LIN {X 0,Y 626.002,Z 844.06,A -85,B 0,C 180,E1 6698.138,E2 6698.138} C_VEL
LIN {X 0,Y 626.101,Z 844.06,A -85,B 0,C 180,E1 6703.663,E2 6703.663} C_VEL
LIN {X 0,Y 628.264,Z 852.739,A -85,B 0,C 180,E1 6704.183,E2 6704.183} C_VEL
LIN {X 0,Y 630.269,Z 865.489,A -85,B 0,C 180,E1 6704.573,E2 6704.573} C_VEL
LIN {X 0,Y 651.429,Z 905.185,A -85,B 0,C 180,E1 6707.05,E2 6707.05} C_VEL
LIN {X 0,Y 646.579,Z 984.33,A -85,B 0,C 180,E1 6708.978,E2 6708.978} C_VEL
LIN {X 0,Y 639.779,Z 1059.441,A -85,B 0,C 180,E1 6712.384,E2 6712.384} C_VEL
LIN {X 0,Y 632.449,Z 1127.06,A -85,B 0,C 180,E1 6717.105,E2 6717.105} C_VEL
LIN {X 0,Y 626.29,Z 1184.219,A -85,B 0,C 180,E1 6722.849,E2 6722.849} C_VEL
LIN {X 0,Y 621.93,Z 1231.471,A -85,B 0,C 180,E1 6729.651,E2 6729.651} C_VEL
LIN {X 0,Y 619.696,Z 1263.198,A -85,B 0,C 180,E1 6736.556,E2 6736.556} C_VEL
LIN {X 0,Y 619.192,Z 1280.004,A -85,B 0,C 180,E1 6742.684,E2 6742.684} C_VEL
LIN {X 0,Y 619.266,Z 1286.38,A -85,B 0,C 180,E1 6747.895,E2 6747.895} C_VEL
LIN {X 0,Y 619.049,Z 1283.806,A -85,B 0,C 180,E1 6754.919,E2 6754.919} C_VEL
LIN {X 0,Y 619.245,Z 1270.708,A -85,B 0,C 180,E1 6761.153,E2 6761.153} C_VEL
LIN {X 0,Y 620.48,Z 1246.742,A -85,B 0,C 180,E1 6767.407,E2 6767.407} C_VEL
LIN {X 0,Y 623.202,Z 1210.805,A -85,B 0,C 180,E1 6773.673,E2 6773.673} C_VEL
LIN {X 0,Y 628.657,Z 1158.622,A -85,B 0,C 180,E1 6779.994,E2 6779.994} C_VEL
LIN {X 0,Y 635.99,Z 1095.052,A -85,B 0,C 180,E1 6785.36,E2 6785.36} C_VEL
LIN {X 0,Y 643.433,Z 1024.758,A -85,B 0,C 180,E1 6789.381,E2 6789.381} C_VEL
LIN {X 0,Y 649.249,Z 949.588,A -85,B 0,C 180,E1 6792.052,E2 6792.052} C_VEL
LIN {X 0,Y 650.101,Z 899.28,A -85,B 0,C 180,E1 6793.162,E2 6793.162} C_VEL
LIN {X 0,Y 618.004,Z 844.06,A -85,B 0,C 180,E1 6797.103,E2 6797.103} C_VEL
LIN {X 0,Y 618.586,Z 844.06,A -85,B 0,C 180,E1 6805.214,E2 6805.214} C_VEL
LIN {X 0,Y 618.31,Z 844.06,A -85,B 0,C 180,E1 6814.598,E2 6814.598} C_VEL
LIN {X 0,Y 618.343,Z 844.06,A -85,B 0,C 180,E1 6823.636,E2 6823.636} C_VEL
LIN {X 0,Y 618.382,Z 844.06,A -85,B 0,C 180,E1 6832.269,E2 6832.269} C_VEL
LIN {X 0,Y 618.586,Z 844.06,A -85,B 0,C 180,E1 6839.32,E2 6839.32} C_VEL
LIN {X 0,Y 618.554,Z 844.06,A -85,B 0,C 180,E1 6846.805,E2 6846.805} C_VEL
LIN {X 0,Y 618.35,Z 844.06,A -85,B 0,C 180,E1 6854.951,E2 6854.951} C_VEL
LIN {X 0,Y 618.062,Z 844.06,A -85,B 0,C 180,E1 6863.054,E2 6863.054} C_VEL
LIN {X 0,Y 617.97,Z 844.06,A -85,B 0,C 180,E1 6871.883,E2 6871.883} C_VEL
LIN {X 0,Y 617.773,Z 844.06,A -85,B 0,C 180,E1 6880.628,E2 6880.628} C_VEL
LIN {X 0,Y 618.221,Z 845.887,A -85,B 0,C 180,E1 6883.215,E2 6883.215} C_VEL
LIN {X 0,Y 651.122,Z 903.195,A -85,B 0,C 180,E1 6887.124,E2 6887.124} C_VEL
LIN {X 0,Y 646.443,Z 978.639,A -85,B 0,C 180,E1 6889.093,E2 6889.093} C_VEL
LIN {X 0,Y 639.82,Z 1050.163,A -85,B 0,C 180,E1 6892.387,E2 6892.387} C_VEL
LIN {X 0,Y 632.376,Z 1116.636,A -85,B 0,C 180,E1 6897.018,E2 6897.018} C_VEL
LIN {X 0,Y 625.899,Z 1175.076,A -85,B 0,C 180,E1 6902.89,E2 6902.89} C_VEL
LIN {X 0,Y 621.742,Z 1219.649,A -85,B 0,C 180,E1 6909.287,E2 6909.287} C_VEL
LIN {X 0,Y 619.652,Z 1249.811,A -85,B 0,C 180,E1 6915.601,E2 6915.601} C_VEL
LIN {X 0,Y 619.132,Z 1267.73,A -85,B 0,C 180,E1 6921.549,E2 6921.549} C_VEL
LIN {X 0,Y 618.746,Z 1276.413,A -85,B 0,C 180,E1 6927.893,E2 6927.893} C_VEL
LIN {X 0,Y 619.029,Z 1275.319,A -85,B 0,C 180,E1 6933.511,E2 6933.511} C_VEL
LIN {X 0,Y 619.043,Z 1264.068,A -85,B 0,C 180,E1 6939.874,E2 6939.874} C_VEL
LIN {X 0,Y 619.898,Z 1243.034,A -85,B 0,C 180,E1 6945.975,E2 6945.975} C_VEL
LIN {X 0,Y 622.4,Z 1209.021,A -85,B 0,C 180,E1 6952.378,E2 6952.378} C_VEL
LIN {X 0,Y 627.314,Z 1160.484,A -85,B 0,C 180,E1 6958.696,E2 6958.696} C_VEL
LIN {X 0,Y 634.383,Z 1098.839,A -85,B 0,C 180,E1 6964.31,E2 6964.31} C_VEL
LIN {X 0,Y 642.002,Z 1029.13,A -85,B 0,C 180,E1 6968.645,E2 6968.645} C_VEL
LIN {X 0,Y 648.194,Z 955.723,A -85,B 0,C 180,E1 6971.557,E2 6971.557} C_VEL
LIN {X 0,Y 649.534,Z 900.272,A -85,B 0,C 180,E1 6972.971,E2 6972.971} C_VEL
LIN {X 0,Y 618.229,Z 844.06,A -85,B 0,C 180,E1 6976.947,E2 6976.947} C_VEL
LIN {X 0,Y 618.186,Z 844.06,A -85,B 0,C 180,E1 6985.268,E2 6985.268} C_VEL
LIN {X 0,Y 618.232,Z 844.06,A -85,B 0,C 180,E1 6993.554,E2 6993.554} C_VEL
LIN {X 0,Y 618.387,Z 844.06,A -85,B 0,C 180,E1 7002.119,E2 7002.119} C_VEL
LIN {X 0,Y 619.238,Z 844.06,A -85,B 0,C 180,E1 7009.389,E2 7009.389} C_VEL
LIN {X 0,Y 619.236,Z 844.06,A -85,B 0,C 180,E1 7017.871,E2 7017.871} C_VEL
LIN {X 0,Y 618.571,Z 844.06,A -85,B 0,C 180,E1 7026.817,E2 7026.817} C_VEL
LIN {X 0,Y 618.341,Z 844.06,A -85,B 0,C 180,E1 7034.904,E2 7034.904} C_VEL
LIN {X 0,Y 618.093,Z 844.06,A -85,B 0,C 180,E1 7043.061,E2 7043.061} C_VEL
LIN {X 0,Y 618.015,Z 844.06,A -85,B 0,C 180,E1 7051.827,E2 7051.827} C_VEL
LIN {X 0,Y 617.714,Z 844.06,A -85,B 0,C 180,E1 7060.572,E2 7060.572} C_VEL
LIN {X 0,Y 618.172,Z 845.961,A -85,B 0,C 180,E1 7063.102,E2 7063.102} C_VEL
LIN {X 0,Y 630.269,Z 865.489,A -85,B 0,C 180,E1 7064.573,E2 7064.573} C_VEL
LIN {X 0,Y 639.982,Z 896.297,A -85,B 0,C 180,E1 7065.929,E2 7065.929} C_VEL
LIN {X 0,Y 645.504,Z 909.832,A -85,B 0,C 180,E1 7066.642,E2 7066.642} C_VEL
LIN {X 0,Y 640.268,Z 987.254,A -85,B 0,C 180,E1 7068.602,E2 7068.602} C_VEL
LIN {X 0,Y 633.06,Z 1061.429,A -85,B 0,C 180,E1 7072.041,E2 7072.041} C_VEL
LIN {X 0,Y 625.297,Z 1128.203,A -85,B 0,C 180,E1 7076.784,E2 7076.784} C_VEL
LIN {X 0,Y 618.672,Z 1185.973,A -85,B 0,C 180,E1 7082.704,E2 7082.704} C_VEL
LIN {X 0,Y 614.273,Z 1231.129,A -85,B 0,C 180,E1 7089.327,E2 7089.327} C_VEL
LIN {X 0,Y 611.806,Z 1263.197,A -85,B 0,C 180,E1 7096.38,E2 7096.38} C_VEL
LIN {X 0,Y 611.195,Z 1280.147,A -85,B 0,C 180,E1 7102.667,E2 7102.667} C_VEL
LIN {X 0,Y 611.278,Z 1286.38,A -85,B 0,C 180,E1 7107.867,E2 7107.867} C_VEL
LIN {X 0,Y 611.058,Z 1283.803,A -85,B 0,C 180,E1 7114.983,E2 7114.983} C_VEL
LIN {X 0,Y 611.24,Z 1270.149,A -85,B 0,C 180,E1 7121.495,E2 7121.495} C_VEL
LIN {X 0,Y 612.589,Z 1246.769,A -85,B 0,C 180,E1 7127.632,E2 7127.632} C_VEL
LIN {X 0,Y 615.51,Z 1210.805,A -85,B 0,C 180,E1 7133.987,E2 7133.987} C_VEL
LIN {X 0,Y 621.262,Z 1160.127,A -85,B 0,C 180,E1 7140.23,E2 7140.23} C_VEL
LIN {X 0,Y 629.016,Z 1096.867,A -85,B 0,C 180,E1 7145.672,E2 7145.672} C_VEL
LIN {X 0,Y 636.904,Z 1027.182,A -85,B 0,C 180,E1 7149.738,E2 7149.738} C_VEL
LIN {X 0,Y 643.085,Z 952.285,A -85,B 0,C 180,E1 7152.469,E2 7152.469} C_VEL
LIN {X 0,Y 644.166,Z 902.371,A -85,B 0,C 180,E1 7153.604,E2 7153.604} C_VEL
LIN {X 0,Y 610.109,Z 844.06,A -85,B 0,C 180,E1 7157.763,E2 7157.763} C_VEL
LIN {X 0,Y 610.509,Z 844.06,A -85,B 0,C 180,E1 7166.321,E2 7166.321} C_VEL
LIN {X 0,Y 610.219,Z 844.06,A -85,B 0,C 180,E1 7175.109,E2 7175.109} C_VEL
LIN {X 0,Y 610.345,Z 844.06,A -85,B 0,C 180,E1 7183.415,E2 7183.415} C_VEL
LIN {X 0,Y 610.388,Z 844.06,A -85,B 0,C 180,E1 7192.167,E2 7192.167} C_VEL
LIN {X 0,Y 610.587,Z 844.06,A -85,B 0,C 180,E1 7199.311,E2 7199.311} C_VEL
LIN {X 0,Y 610.683,Z 844.06,A -85,B 0,C 180,E1 7206.442,E2 7206.442} C_VEL
LIN {X 0,Y 610.294,Z 844.06,A -85,B 0,C 180,E1 7215.153,E2 7215.153} C_VEL
LIN {X 0,Y 610.144,Z 844.06,A -85,B 0,C 180,E1 7222.693,E2 7222.693} C_VEL
LIN {X 0,Y 610.061,Z 844.06,A -85,B 0,C 180,E1 7230.949,E2 7230.949} C_VEL
LIN {X 0,Y 609.85,Z 844.06,A -85,B 0,C 180,E1 7239.4,E2 7239.4} C_VEL
LIN {X 0,Y 610.054,Z 845.695,A -85,B 0,C 180,E1 7242.388,E2 7242.388} C_VEL
LIN {X 0,Y 644.996,Z 906.338,A -85,B 0,C 180,E1 7246.69,E2 7246.69} C_VEL
LIN {X 0,Y 640.096,Z 981.944,A -85,B 0,C 180,E1 7248.736,E2 7248.736} C_VEL
LIN {X 0,Y 632.886,Z 1053.967,A -85,B 0,C 180,E1 7252.147,E2 7252.147} C_VEL
LIN {X 0,Y 624.872,Z 1120.556,A -85,B 0,C 180,E1 7256.926,E2 7256.926} C_VEL
LIN {X 0,Y 617.979,Z 1178.841,A -85,B 0,C 180,E1 7263,E2 7263} C_VEL
LIN {X 0,Y 613.578,Z 1223.371,A -85,B 0,C 180,E1 7269.673,E2 7269.673} C_VEL
LIN {X 0,Y 611.531,Z 1252.307,A -85,B 0,C 180,E1 7276.085,E2 7276.085} C_VEL
LIN {X 0,Y 611.009,Z 1269.257,A -85,B 0,C 180,E1 7282.154,E2 7282.154} C_VEL
LIN {X 0,Y 610.752,Z 1276.413,A -85,B 0,C 180,E1 7287.866,E2 7287.866} C_VEL
LIN {X 0,Y 611.052,Z 1275.32,A -85,B 0,C 180,E1 7293.557,E2 7293.557} C_VEL
LIN {X 0,Y 611.058,Z 1264.069,A -85,B 0,C 180,E1 7300.005,E2 7300.005} C_VEL
LIN {X 0,Y 611.996,Z 1243.038,A -85,B 0,C 180,E1 7306.187,E2 7306.187} C_VEL
LIN {X 0,Y 614.716,Z 1209.023,A -85,B 0,C 180,E1 7312.673,E2 7312.673} C_VEL
LIN {X 0,Y 619.887,Z 1161.231,A -85,B 0,C 180,E1 7318.988,E2 7318.988} C_VEL
LIN {X 0,Y 627.318,Z 1100.446,A -85,B 0,C 180,E1 7324.619,E2 7324.619} C_VEL
LIN {X 0,Y 635.357,Z 1031.58,A -85,B 0,C 180,E1 7328.985,E2 7328.985} C_VEL
LIN {X 0,Y 641.984,Z 958.36,A -85,B 0,C 180,E1 7331.959,E2 7331.959} C_VEL
LIN {X 0,Y 643.686,Z 903.738,A -85,B 0,C 180,E1 7333.39,E2 7333.39} C_VEL
LIN {X 0,Y 610.146,Z 844.06,A -85,B 0,C 180,E1 7337.638,E2 7337.638} C_VEL
LIN {X 0,Y 610.15,Z 844.06,A -85,B 0,C 180,E1 7346.372,E2 7346.372} C_VEL
LIN {X 0,Y 610.27,Z 844.06,A -85,B 0,C 180,E1 7355.099,E2 7355.099} C_VEL
LIN {X 0,Y 610.582,Z 844.06,A -85,B 0,C 180,E1 7363.374,E2 7363.374} C_VEL
LIN {X 0,Y 610.862,Z 844.06,A -85,B 0,C 180,E1 7370.687,E2 7370.687} C_VEL
LIN {X 0,Y 611.253,Z 844.06,A -85,B 0,C 180,E1 7377.843,E2 7377.843} C_VEL
LIN {X 0,Y 610.695,Z 844.06,A -85,B 0,C 180,E1 7386.395,E2 7386.395} C_VEL
LIN {X 0,Y 610.29,Z 844.06,A -85,B 0,C 180,E1 7395.106,E2 7395.106} C_VEL
LIN {X 0,Y 610.163,Z 844.06,A -85,B 0,C 180,E1 7402.642,E2 7402.642} C_VEL
LIN {X 0,Y 610.075,Z 844.06,A -85,B 0,C 180,E1 7410.951,E2 7410.951} C_VEL
LIN {X 0,Y 609.814,Z 844.06,A -85,B 0,C 180,E1 7419.343,E2 7419.343} C_VEL
LIN {X 0,Y 609.982,Z 845.677,A -85,B 0,C 180,E1 7422.271,E2 7422.271} C_VEL
LIN {X 0,Y 639.982,Z 896.297,A -85,B 0,C 180,E1 7425.929,E2 7425.929} C_VEL
LIN {X 0,Y 641.79,Z 912.839,A -85,B 0,C 180,E1 7426.384,E2 7426.384} C_VEL
LIN {X 0,Y 638.723,Z 931.558,A -85,B 0,C 180,E1 7426.567,E2 7426.567} C_VEL
LIN {X 0,Y 633.009,Z 1002.704,A -85,B 0,C 180,E1 7428.723,E2 7428.723} C_VEL
LIN {X 0,Y 625.002,Z 1075.016,A -85,B 0,C 180,E1 7432.413,E2 7432.413} C_VEL
LIN {X 0,Y 616.67,Z 1140.57,A -85,B 0,C 180,E1 7437.469,E2 7437.469} C_VEL
LIN {X 0,Y 609.846,Z 1195.877,A -85,B 0,C 180,E1 7443.613,E2 7443.613} C_VEL
LIN {X 0,Y 605.6,Z 1237.509,A -85,B 0,C 180,E1 7450.241,E2 7450.241} C_VEL
LIN {X 0,Y 603.548,Z 1265.683,A -85,B 0,C 180,E1 7456.93,E2 7456.93} C_VEL
LIN {X 0,Y 602.957,Z 1281.732,A -85,B 0,C 180,E1 7463.501,E2 7463.501} C_VEL
LIN {X 0,Y 602.724,Z 1286.838,A -85,B 0,C 180,E1 7469.279,E2 7469.279} C_VEL
LIN {X 0,Y 602.912,Z 1282.883,A -85,B 0,C 180,E1 7475.774,E2 7475.774} C_VEL
LIN {X 0,Y 603.311,Z 1267.998,A -85,B 0,C 180,E1 7482.337,E2 7482.337} C_VEL
LIN {X 0,Y 604.879,Z 1243.162,A -85,B 0,C 180,E1 7488.643,E2 7488.643} C_VEL
LIN {X 0,Y 608.656,Z 1204.137,A -85,B 0,C 180,E1 7495.263,E2 7495.263} C_VEL
LIN {X 0,Y 615.213,Z 1150.124,A -85,B 0,C 180,E1 7501.632,E2 7501.632} C_VEL
LIN {X 0,Y 623.548,Z 1086.517,A -85,B 0,C 180,E1 7506.84,E2 7506.84} C_VEL
LIN {X 0,Y 631.633,Z 1017.29,A -85,B 0,C 180,E1 7510.659,E2 7510.659} C_VEL
LIN {X 0,Y 637.609,Z 945.851,A -85,B 0,C 180,E1 7513.112,E2 7513.112} C_VEL
LIN {X 0,Y 638.224,Z 905.427,A -85,B 0,C 180,E1 7514.057,E2 7514.057} C_VEL
LIN {X 0,Y 602.173,Z 844.06,A -85,B 0,C 180,E1 7518.668,E2 7518.668} C_VEL
LIN {X 0,Y 602.414,Z 844.06,A -85,B 0,C 180,E1 7527.494,E2 7527.494} C_VEL
LIN {X 0,Y 602.18,Z 844.06,A -85,B 0,C 180,E1 7535.464,E2 7535.464} C_VEL
LIN {X 0,Y 602.389,Z 844.06,A -85,B 0,C 180,E1 7543.19,E2 7543.19} C_VEL
LIN {X 0,Y 602.394,Z 844.06,A -85,B 0,C 180,E1 7552.062,E2 7552.062} C_VEL
LIN {X 0,Y 602.588,Z 844.06,A -85,B 0,C 180,E1 7559.302,E2 7559.302} C_VEL
LIN {X 0,Y 602.663,Z 844.06,A -85,B 0,C 180,E1 7566.528,E2 7566.528} C_VEL
LIN {X 0,Y 602.255,Z 844.06,A -85,B 0,C 180,E1 7575.361,E2 7575.361} C_VEL
LIN {X 0,Y 602.039,Z 844.06,A -85,B 0,C 180,E1 7583.157,E2 7583.157} C_VEL
LIN {X 0,Y 602.055,Z 844.06,A -85,B 0,C 180,E1 7591.128,E2 7591.128} C_VEL
LIN {X 0,Y 601.8,Z 844.06,A -85,B 0,C 180,E1 7600.032,E2 7600.032} C_VEL
LIN {X 0,Y 601.985,Z 845.823,A -85,B 0,C 180,E1 7601.541,E2 7601.541} C_VEL
LIN {X 0,Y 638.637,Z 908.901,A -85,B 0,C 180,E1 7606.213,E2 7606.213} C_VEL
LIN {X 0,Y 633.546,Z 986.704,A -85,B 0,C 180,E1 7608.44,E2 7608.44} C_VEL
LIN {X 0,Y 625.816,Z 1058.298,A -85,B 0,C 180,E1 7611.946,E2 7611.946} C_VEL
LIN {X 0,Y 617.375,Z 1124.269,A -85,B 0,C 180,E1 7616.839,E2 7616.839} C_VEL
LIN {X 0,Y 610.298,Z 1180.481,A -85,B 0,C 180,E1 7622.854,E2 7622.854} C_VEL
LIN {X 0,Y 605.653,Z 1224.708,A -85,B 0,C 180,E1 7629.654,E2 7629.654} C_VEL
LIN {X 0,Y 603.532,Z 1253.36,A -85,B 0,C 180,E1 7636.189,E2 7636.189} C_VEL
LIN {X 0,Y 602.998,Z 1270.597,A -85,B 0,C 180,E1 7642.776,E2 7642.776} C_VEL
LIN {X 0,Y 602.834,Z 1276.848,A -85,B 0,C 180,E1 7649.279,E2 7649.279} C_VEL
LIN {X 0,Y 603.349,Z 1272.815,A -85,B 0,C 180,E1 7655.77,E2 7655.77} C_VEL
LIN {X 0,Y 604.141,Z 1254.369,A -85,B 0,C 180,E1 7663.427,E2 7663.427} C_VEL
LIN {X 0,Y 606.173,Z 1220.954,A -85,B 0,C 180,E1 7670.948,E2 7670.948} C_VEL
LIN {X 0,Y 610.986,Z 1174.739,A -85,B 0,C 180,E1 7677.778,E2 7677.778} C_VEL
LIN {X 0,Y 618.492,Z 1116.109,A -85,B 0,C 180,E1 7683.777,E2 7683.777} C_VEL
LIN {X 0,Y 626.996,Z 1048.85,A -85,B 0,C 180,E1 7688.515,E2 7688.515} C_VEL
LIN {X 0,Y 634.3,Z 974.856,A -85,B 0,C 180,E1 7691.928,E2 7691.928} C_VEL
LIN {X 0,Y 637.711,Z 906.961,A -85,B 0,C 180,E1 7693.823,E2 7693.823} C_VEL
LIN {X 0,Y 603.496,Z 848.586,A -85,B 0,C 180,E1 7698.159,E2 7698.159} C_VEL
LIN {X 0,Y 602.067,Z 844.06,A -85,B 0,C 180,E1 7698.693,E2 7698.693} C_VEL
LIN {X 0,Y 602.188,Z 844.06,A -85,B 0,C 180,E1 7707.528,E2 7707.528} C_VEL
LIN {X 0,Y 602.45,Z 844.06,A -85,B 0,C 180,E1 7717.001,E2 7717.001} C_VEL
LIN {X 0,Y 603.091,Z 844.06,A -85,B 0,C 180,E1 7726.15,E2 7726.15} C_VEL
LIN {X 0,Y 602.563,Z 844.06,A -85,B 0,C 180,E1 7734.921,E2 7734.921} C_VEL
LIN {X 0,Y 602.486,Z 844.06,A -85,B 0,C 180,E1 7742.141,E2 7742.141} C_VEL
LIN {X 0,Y 602.347,Z 844.06,A -85,B 0,C 180,E1 7749.398,E2 7749.398} C_VEL
LIN {X 0,Y 602.15,Z 844.06,A -85,B 0,C 180,E1 7756.817,E2 7756.817} C_VEL
LIN {X 0,Y 601.982,Z 844.06,A -85,B 0,C 180,E1 7764.545,E2 7764.545} C_VEL
LIN {X 0,Y 601.966,Z 844.06,A -85,B 0,C 180,E1 7772.78,E2 7772.78} C_VEL
LIN {X 0,Y 601.834,Z 845.482,A -85,B 0,C 180,E1 7781.41,E2 7781.41} C_VEL
LIN {X 0,Y 639.487,Z 909.82,A -85,B 0,C 180,E1 7786.131,E2 7786.131} C_VEL
LIN {X 0,Y 638.723,Z 931.558,A -85,B 0,C 180,E1 7786.567,E2 7786.567} C_VEL
LIN {X 0,Y 630.191,Z 965.784,A -85,B 0,C 180,E1 7786.932,E2 7786.932} C_VEL
LIN {X 0,Y 622.808,Z 1040.446,A -85,B 0,C 180,E1 7789.96,E2 7789.96} C_VEL
LIN {X 0,Y 613.795,Z 1109.857,A -85,B 0,C 180,E1 7794.409,E2 7794.409} C_VEL
LIN {X 0,Y 605.326,Z 1171.403,A -85,B 0,C 180,E1 7800.22,E2 7800.22} C_VEL
LIN {X 0,Y 599.48,Z 1220.506,A -85,B 0,C 180,E1 7806.914,E2 7806.914} C_VEL
LIN {X 0,Y 596.496,Z 1256.298,A -85,B 0,C 180,E1 7814.139,E2 7814.139} C_VEL
LIN {X 0,Y 595.561,Z 1277.621,A -85,B 0,C 180,E1 7821.212,E2 7821.212} C_VEL
LIN {X 0,Y 595.276,Z 1286.38,A -85,B 0,C 180,E1 7827.81,E2 7827.81} C_VEL
LIN {X 0,Y 595.034,Z 1283.798,A -85,B 0,C 180,E1 7835.118,E2 7835.118} C_VEL
LIN {X 0,Y 595.261,Z 1270.096,A -85,B 0,C 180,E1 7841.824,E2 7841.824} C_VEL
LIN {X 0,Y 596.849,Z 1246.047,A -85,B 0,C 180,E1 7848.271,E2 7848.271} C_VEL
LIN {X 0,Y 600.598,Z 1208.153,A -85,B 0,C 180,E1 7855.021,E2 7855.021} C_VEL
LIN {X 0,Y 607.323,Z 1156.087,A -85,B 0,C 180,E1 7861.439,E2 7861.439} C_VEL
LIN {X 0,Y 616.062,Z 1092.607,A -85,B 0,C 180,E1 7866.879,E2 7866.879} C_VEL
LIN {X 0,Y 624.759,Z 1023.36,A -85,B 0,C 180,E1 7870.876,E2 7870.876} C_VEL
LIN {X 0,Y 631.511,Z 949.245,A -85,B 0,C 180,E1 7873.53,E2 7873.53} C_VEL
LIN {X 0,Y 632.398,Z 908.725,A -85,B 0,C 180,E1 7874.508,E2 7874.508} C_VEL
LIN {X 0,Y 594.26,Z 844.06,A -85,B 0,C 180,E1 7879.65,E2 7879.65} C_VEL
LIN {X 0,Y 594.331,Z 844.06,A -85,B 0,C 180,E1 7888.739,E2 7888.739} C_VEL
LIN {X 0,Y 594.029,Z 844.06,A -85,B 0,C 180,E1 7896.708,E2 7896.708} C_VEL
LIN {X 0,Y 594.166,Z 844.06,A -85,B 0,C 180,E1 7904.474,E2 7904.474} C_VEL
LIN {X 0,Y 594.399,Z 844.06,A -85,B 0,C 180,E1 7911.955,E2 7911.955} C_VEL
LIN {X 0,Y 594.6,Z 844.06,A -85,B 0,C 180,E1 7919.293,E2 7919.293} C_VEL
LIN {X 0,Y 594.626,Z 844.06,A -85,B 0,C 180,E1 7926.616,E2 7926.616} C_VEL
LIN {X 0,Y 594.213,Z 844.06,A -85,B 0,C 180,E1 7935.574,E2 7935.574} C_VEL
LIN {X 0,Y 594.014,Z 844.06,A -85,B 0,C 180,E1 7943.345,E2 7943.345} C_VEL
LIN {X 0,Y 593.988,Z 844.06,A -85,B 0,C 180,E1 7951.599,E2 7951.599} C_VEL
LIN {X 0,Y 593.788,Z 844.737,A -85,B 0,C 180,E1 7960.619,E2 7960.619} C_VEL
LIN {X 0,Y 631.903,Z 910.624,A -85,B 0,C 180,E1 7965.667,E2 7965.667} C_VEL
LIN {X 0,Y 627.171,Z 989.671,A -85,B 0,C 180,E1 7968.064,E2 7968.064} C_VEL
LIN {X 0,Y 618.902,Z 1061.446,A -85,B 0,C 180,E1 7971.673,E2 7971.673} C_VEL
LIN {X 0,Y 609.783,Z 1128.357,A -85,B 0,C 180,E1 7976.787,E2 7976.787} C_VEL
LIN {X 0,Y 602.362,Z 1184.134,A -85,B 0,C 180,E1 7982.974,E2 7982.974} C_VEL
LIN {X 0,Y 597.785,Z 1225.778,A -85,B 0,C 180,E1 7989.584,E2 7989.584} C_VEL
LIN {X 0,Y 595.521,Z 1254.664,A -85,B 0,C 180,E1 7996.376,E2 7996.376} C_VEL
LIN {X 0,Y 595.012,Z 1270.593,A -85,B 0,C 180,E1 8002.679,E2 8002.679} C_VEL
LIN {X 0,Y 594.855,Z 1276.848,A -85,B 0,C 180,E1 8009.27,E2 8009.27} C_VEL
LIN {X 0,Y 595.372,Z 1272.905,A -85,B 0,C 180,E1 8015.785,E2 8015.785} C_VEL
LIN {X 0,Y 596.161,Z 1254.37,A -85,B 0,C 180,E1 8023.61,E2 8023.61} C_VEL
LIN {X 0,Y 598.335,Z 1221.307,A -85,B 0,C 180,E1 8031.173,E2 8031.173} C_VEL
LIN {X 0,Y 603.513,Z 1175.31,A -85,B 0,C 180,E1 8038.08,E2 8038.08} C_VEL
LIN {X 0,Y 611.38,Z 1117.449,A -85,B 0,C 180,E1 8044.1,E2 8044.1} C_VEL
LIN {X 0,Y 620.389,Z 1050.271,A -85,B 0,C 180,E1 8048.909,E2 8048.909} C_VEL
LIN {X 0,Y 628.192,Z 975.916,A -85,B 0,C 180,E1 8052.387,E2 8052.387} C_VEL
LIN {X 0,Y 631.865,Z 910.539,A -85,B 0,C 180,E1 8054.249,E2 8054.249} C_VEL
LIN {X 0,Y 597.028,Z 850.282,A -85,B 0,C 180,E1 8058.829,E2 8058.829} C_VEL
LIN {X 0,Y 594.037,Z 844.06,A -85,B 0,C 180,E1 8059.336,E2 8059.336} C_VEL
LIN {X 0,Y 594.214,Z 844.06,A -85,B 0,C 180,E1 8068.414,E2 8068.414} C_VEL
LIN {X 0,Y 594.431,Z 844.06,A -85,B 0,C 180,E1 8076.673,E2 8076.673} C_VEL
LIN {X 0,Y 595.06,Z 844.06,A -85,B 0,C 180,E1 8085.96,E2 8085.96} C_VEL
LIN {X 0,Y 594.555,Z 844.06,A -85,B 0,C 180,E1 8094.853,E2 8094.853} C_VEL
LIN {X 0,Y 594.497,Z 844.06,A -85,B 0,C 180,E1 8102.17,E2 8102.17} C_VEL
LIN {X 0,Y 594.351,Z 844.06,A -85,B 0,C 180,E1 8109.526,E2 8109.526} C_VEL
LIN {X 0,Y 594.166,Z 844.06,A -85,B 0,C 180,E1 8117.05,E2 8117.05} C_VEL
LIN {X 0,Y 593.955,Z 844.06,A -85,B 0,C 180,E1 8124.985,E2 8124.985} C_VEL
LIN {X 0,Y 593.904,Z 844.06,A -85,B 0,C 180,E1 8133.283,E2 8133.283} C_VEL
LIN {X 0,Y 593.96,Z 846.045,A -85,B 0,C 180,E1 8140.554,E2 8140.554} C_VEL
LIN {X 0,Y 631.597,Z 909.164,A -85,B 0,C 180,E1 8145.429,E2 8145.429} C_VEL
LIN {X 0,Y 633.352,Z 922.085,A -85,B 0,C 180,E1 8145.877,E2 8145.877} C_VEL
LIN {X 0,Y 630.191,Z 965.784,A -85,B 0,C 180,E1 8146.932,E2 8146.932} C_VEL
LIN {X 0,Y 621.085,Z 999.235,A -85,B 0,C 180,E1 8147.582,E2 8147.582} C_VEL
LIN {X 0,Y 612.174,Z 1072.89,A -85,B 0,C 180,E1 8151.327,E2 8151.327} C_VEL
LIN {X 0,Y 602.922,Z 1138.686,A -85,B 0,C 180,E1 8156.439,E2 8156.439} C_VEL
LIN {X 0,Y 595.243,Z 1194.536,A -85,B 0,C 180,E1 8162.726,E2 8162.726} C_VEL
LIN {X 0,Y 590.122,Z 1237.505,A -85,B 0,C 180,E1 8169.7,E2 8169.7} C_VEL
LIN {X 0,Y 587.589,Z 1266.845,A -85,B 0,C 180,E1 8176.948,E2 8176.948} C_VEL
LIN {X 0,Y 586.963,Z 1282.869,A -85,B 0,C 180,E1 8184.059,E2 8184.059} C_VEL
LIN {X 0,Y 586.597,Z 1286.838,A -85,B 0,C 180,E1 8190.741,E2 8190.741} C_VEL
LIN {X 0,Y 586.966,Z 1281.727,A -85,B 0,C 180,E1 8196.677,E2 8196.677} C_VEL
LIN {X 0,Y 587.825,Z 1264.523,A -85,B 0,C 180,E1 8203.806,E2 8203.806} C_VEL
LIN {X 0,Y 590.982,Z 1231.552,A -85,B 0,C 180,E1 8211.449,E2 8211.449} C_VEL
LIN {X 0,Y 596.367,Z 1185.929,A -85,B 0,C 180,E1 8218.413,E2 8218.413} C_VEL
LIN {X 0,Y 604.488,Z 1127.965,A -85,B 0,C 180,E1 8224.541,E2 8224.541} C_VEL
LIN {X 0,Y 613.812,Z 1060.538,A -85,B 0,C 180,E1 8229.434,E2 8229.434} C_VEL
LIN {X 0,Y 622.441,Z 986.1,A -85,B 0,C 180,E1 8232.909,E2 8232.909} C_VEL
LIN {X 0,Y 626.686,Z 912.291,A -85,B 0,C 180,E1 8234.955,E2 8234.955} C_VEL
LIN {X 0,Y 586.267,Z 844.06,A -85,B 0,C 180,E1 8240.471,E2 8240.471} C_VEL
LIN {X 0,Y 586.285,Z 844.06,A -85,B 0,C 180,E1 8247.993,E2 8247.993} C_VEL
LIN {X 0,Y 586.026,Z 844.06,A -85,B 0,C 180,E1 8256.734,E2 8256.734} C_VEL
LIN {X 0,Y 586.182,Z 844.06,A -85,B 0,C 180,E1 8264.257,E2 8264.257} C_VEL
LIN {X 0,Y 586.419,Z 844.06,A -85,B 0,C 180,E1 8271.844,E2 8271.844} C_VEL
LIN {X 0,Y 586.601,Z 844.06,A -85,B 0,C 180,E1 8279.283,E2 8279.283} C_VEL
LIN {X 0,Y 586.613,Z 844.06,A -85,B 0,C 180,E1 8286.707,E2 8286.707} C_VEL
LIN {X 0,Y 586.46,Z 844.06,A -85,B 0,C 180,E1 8294.25,E2 8294.25} C_VEL
LIN {X 0,Y 586.025,Z 844.06,A -85,B 0,C 180,E1 8303.266,E2 8303.266} C_VEL
LIN {X 0,Y 585.905,Z 844.06,A -85,B 0,C 180,E1 8312.087,E2 8312.087} C_VEL
LIN {X 0,Y 585.929,Z 845.473,A -85,B 0,C 180,E1 8319.727,E2 8319.727} C_VEL
LIN {X 0,Y 623.732,Z 909.084,A -85,B 0,C 180,E1 8324.888,E2 8324.888} C_VEL
LIN {X 0,Y 627.011,Z 921.583,A -85,B 0,C 180,E1 8325.499,E2 8325.499} C_VEL
LIN {X 0,Y 620.96,Z 991.443,A -85,B 0,C 180,E1 8327.634,E2 8327.634} C_VEL
LIN {X 0,Y 612.352,Z 1062.034,A -85,B 0,C 180,E1 8331.231,E2 8331.231} C_VEL
LIN {X 0,Y 602.741,Z 1128.788,A -85,B 0,C 180,E1 8336.393,E2 8336.393} C_VEL
LIN {X 0,Y 594.859,Z 1184.695,A -85,B 0,C 180,E1 8342.684,E2 8342.684} C_VEL
LIN {X 0,Y 590.017,Z 1225.773,A -85,B 0,C 180,E1 8349.303,E2 8349.303} C_VEL
LIN {X 0,Y 587.578,Z 1254.663,A -85,B 0,C 180,E1 8356.188,E2 8356.188} C_VEL
LIN {X 0,Y 587.03,Z 1270.589,A -85,B 0,C 180,E1 8362.578,E2 8362.578} C_VEL
LIN {X 0,Y 586.853,Z 1276.848,A -85,B 0,C 180,E1 8369.26,E2 8369.26} C_VEL
LIN {X 0,Y 587.386,Z 1272.894,A -85,B 0,C 180,E1 8375.873,E2 8375.873} C_VEL
LIN {X 0,Y 588.155,Z 1254.372,A -85,B 0,C 180,E1 8383.799,E2 8383.799} C_VEL
LIN {X 0,Y 590.474,Z 1222.359,A -85,B 0,C 180,E1 8391.271,E2 8391.271} C_VEL
LIN {X 0,Y 595.942,Z 1176.92,A -85,B 0,C 180,E1 8398.261,E2 8398.261} C_VEL
LIN {X 0,Y 604.211,Z 1119.325,A -85,B 0,C 180,E1 8404.384,E2 8404.384} C_VEL
LIN {X 0,Y 613.75,Z 1052.329,A -85,B 0,C 180,E1 8409.273,E2 8409.273} C_VEL
LIN {X 0,Y 622.012,Z 978.323,A -85,B 0,C 180,E1 8412.807,E2 8412.807} C_VEL
LIN {X 0,Y 625.949,Z 913.829,A -85,B 0,C 180,E1 8414.7,E2 8414.7} C_VEL
LIN {X 0,Y 592.883,Z 856.335,A -85,B 0,C 180,E1 8419.181,E2 8419.181} C_VEL
LIN {X 0,Y 586.013,Z 844.06,A -85,B 0,C 180,E1 8420.215,E2 8420.215} C_VEL
LIN {X 0,Y 586.197,Z 844.06,A -85,B 0,C 180,E1 8429.664,E2 8429.664} C_VEL
LIN {X 0,Y 586.413,Z 844.06,A -85,B 0,C 180,E1 8437.943,E2 8437.943} C_VEL
LIN {X 0,Y 587.197,Z 844.06,A -85,B 0,C 180,E1 8447.29,E2 8447.29} C_VEL
LIN {X 0,Y 587.239,Z 844.06,A -85,B 0,C 180,E1 8457.755,E2 8457.755} C_VEL
LIN {X 0,Y 586.612,Z 844.06,A -85,B 0,C 180,E1 8466.659,E2 8466.659} C_VEL
LIN {X 0,Y 586.456,Z 844.06,A -85,B 0,C 180,E1 8474.201,E2 8474.201} C_VEL
LIN {X 0,Y 586.058,Z 844.06,A -85,B 0,C 180,E1 8483.273,E2 8483.273} C_VEL
LIN {X 0,Y 585.934,Z 844.06,A -85,B 0,C 180,E1 8492.028,E2 8492.028} C_VEL
LIN {X 0,Y 585.942,Z 845.776,A -85,B 0,C 180,E1 8499.627,E2 8499.627} C_VEL
LIN {X 0,Y 624.283,Z 909.609,A -85,B 0,C 180,E1 8504.774,E2 8504.774} C_VEL
LIN {X 0,Y 627.676,Z 920.77,A -85,B 0,C 180,E1 8505.342,E2 8505.342} C_VEL
LIN {X 0,Y 621.239,Z 997.597,A -85,B 0,C 180,E1 8507.516,E2 8507.516} C_VEL
LIN {X 0,Y 621.085,Z 999.235,A -85,B 0,C 180,E1 8507.582,E2 8507.582} C_VEL
LIN {X 0,Y 611.443,Z 1031.876,A -85,B 0,C 180,E1 8508.529,E2 8508.529} C_VEL
LIN {X 0,Y 601.794,Z 1100.442,A -85,B 0,C 180,E1 8512.749,E2 8512.749} C_VEL
LIN {X 0,Y 592.022,Z 1163.121,A -85,B 0,C 180,E1 8518.471,E2 8518.471} C_VEL
LIN {X 0,Y 584.905,Z 1213.217,A -85,B 0,C 180,E1 8525.073,E2 8525.073} C_VEL
LIN {X 0,Y 580.959,Z 1248.31,A -85,B 0,C 180,E1 8531.724,E2 8531.724} C_VEL
LIN {X 0,Y 579.294,Z 1270.293,A -85,B 0,C 180,E1 8537.911,E2 8537.911} C_VEL
LIN {X 0,Y 578.941,Z 1283.791,A -85,B 0,C 180,E1 8544.74,E2 8544.74} C_VEL
LIN {X 0,Y 578.619,Z 1286.838,A -85,B 0,C 180,E1 8550.751,E2 8550.751} C_VEL
LIN {X 0,Y 579.174,Z 1280.513,A -85,B 0,C 180,E1 8557.523,E2 8557.523} C_VEL
LIN {X 0,Y 580.698,Z 1259.227,A -85,B 0,C 180,E1 8565.509,E2 8565.509} C_VEL
LIN {X 0,Y 583.835,Z 1223.742,A -85,B 0,C 180,E1 8573.167,E2 8573.167} C_VEL
LIN {X 0,Y 590.374,Z 1174.488,A -85,B 0,C 180,E1 8580.233,E2 8580.233} C_VEL
LIN {X 0,Y 599.593,Z 1114.992,A -85,B 0,C 180,E1 8586.111,E2 8586.111} C_VEL
LIN {X 0,Y 609.541,Z 1046.195,A -85,B 0,C 180,E1 8590.739,E2 8590.739} C_VEL
LIN {X 0,Y 617.837,Z 970.224,A -85,B 0,C 180,E1 8593.978,E2 8593.978} C_VEL
LIN {X 0,Y 620.662,Z 915.37,A -85,B 0,C 180,E1 8595.435,E2 8595.435} C_VEL
LIN {X 0,Y 578.251,Z 844.06,A -85,B 0,C 180,E1 8601.46,E2 8601.46} C_VEL
LIN {X 0,Y 578.229,Z 844.06,A -85,B 0,C 180,E1 8609.258,E2 8609.258} C_VEL
LIN {X 0,Y 578.014,Z 844.06,A -85,B 0,C 180,E1 8618.656,E2 8618.656} C_VEL
LIN {X 0,Y 578.317,Z 844.06,A -85,B 0,C 180,E1 8627.141,E2 8627.141} C_VEL
LIN {X 0,Y 579.072,Z 844.06,A -85,B 0,C 180,E1 8636.269,E2 8636.269} C_VEL
LIN {X 0,Y 579.011,Z 844.06,A -85,B 0,C 180,E1 8645.286,E2 8645.286} C_VEL
LIN {X 0,Y 578.399,Z 844.06,A -85,B 0,C 180,E1 8654.453,E2 8654.453} C_VEL
LIN {X 0,Y 578.091,Z 844.06,A -85,B 0,C 180,E1 8662.392,E2 8662.392} C_VEL
LIN {X 0,Y 577.917,Z 844.06,A -85,B 0,C 180,E1 8671.478,E2 8671.478} C_VEL
LIN {X 0,Y 578.015,Z 845.963,A -85,B 0,C 180,E1 8678.781,E2 8678.781} C_VEL
LIN {X 0,Y 616.663,Z 909.758,A -85,B 0,C 180,E1 8684.241,E2 8684.241} C_VEL
LIN {X 0,Y 621.15,Z 924.07,A -85,B 0,C 180,E1 8685.033,E2 8685.033} C_VEL
LIN {X 0,Y 614.582,Z 995.067,A -85,B 0,C 180,E1 8687.267,E2 8687.267} C_VEL
LIN {X 0,Y 605.368,Z 1065.77,A -85,B 0,C 180,E1 8690.98,E2 8690.98} C_VEL
LIN {X 0,Y 595.425,Z 1131.118,A -85,B 0,C 180,E1 8696.168,E2 8696.168} C_VEL
LIN {X 0,Y 587.208,Z 1186.149,A -85,B 0,C 180,E1 8702.507,E2 8702.507} C_VEL
LIN {X 0,Y 582.011,Z 1227.72,A -85,B 0,C 180,E1 8709.405,E2 8709.405} C_VEL
LIN {X 0,Y 579.583,Z 1255.823,A -85,B 0,C 180,E1 8716.379,E2 8716.379} C_VEL
LIN {X 0,Y 579.047,Z 1271.797,A -85,B 0,C 180,E1 8723.232,E2 8723.232} C_VEL
LIN {X 0,Y 579.365,Z 1276.827,A -85,B 0,C 180,E1 8730.75,E2 8730.75} C_VEL
LIN {X 0,Y 579.292,Z 1269.075,A -85,B 0,C 180,E1 8738.279,E2 8738.279} C_VEL
LIN {X 0,Y 580.077,Z 1249.006,A -85,B 0,C 180,E1 8745.544,E2 8745.544} C_VEL
LIN {X 0,Y 583.005,Z 1217.526,A -85,B 0,C 180,E1 8752.458,E2 8752.458} C_VEL
LIN {X 0,Y 589.101,Z 1172.212,A -85,B 0,C 180,E1 8759.24,E2 8759.24} C_VEL
LIN {X 0,Y 598.335,Z 1112.27,A -85,B 0,C 180,E1 8765.45,E2 8765.45} C_VEL
LIN {X 0,Y 608.407,Z 1044.81,A -85,B 0,C 180,E1 8770.2,E2 8770.2} C_VEL
LIN {X 0,Y 617.05,Z 970.333,A -85,B 0,C 180,E1 8773.586,E2 8773.586} C_VEL
LIN {X 0,Y 620,Z 916.735,A -85,B 0,C 180,E1 8775.176,E2 8775.176} C_VEL
LIN {X 0,Y 587.451,Z 860.426,A -85,B 0,C 180,E1 8779.724,E2 8779.724} C_VEL
LIN {X 0,Y 577.984,Z 844.06,A -85,B 0,C 180,E1 8781.311,E2 8781.311} C_VEL
LIN {X 0,Y 578.205,Z 844.06,A -85,B 0,C 180,E1 8790.935,E2 8790.935} C_VEL
LIN {X 0,Y 578.324,Z 844.06,A -85,B 0,C 180,E1 8799.234,E2 8799.234} C_VEL
LIN {X 0,Y 579.23,Z 844.06,A -85,B 0,C 180,E1 8808.647,E2 8808.647} C_VEL
LIN {X 0,Y 579.244,Z 844.06,A -85,B 0,C 180,E1 8817.724,E2 8817.724} C_VEL
LIN {X 0,Y 578.579,Z 844.06,A -85,B 0,C 180,E1 8826.752,E2 8826.752} C_VEL
LIN {X 0,Y 578.394,Z 844.06,A -85,B 0,C 180,E1 8834.403,E2 8834.403} C_VEL
LIN {X 0,Y 578.148,Z 844.06,A -85,B 0,C 180,E1 8842.337,E2 8842.337} C_VEL
LIN {X 0,Y 577.951,Z 844.06,A -85,B 0,C 180,E1 8851.483,E2 8851.483} C_VEL
LIN {X 0,Y 577.874,Z 845.426,A -85,B 0,C 180,E1 8858.648,E2 8858.648} C_VEL
LIN {X 0,Y 618.326,Z 912.425,A -85,B 0,C 180,E1 8864.272,E2 8864.272} C_VEL
LIN {X 0,Y 621.775,Z 924.263,A -85,B 0,C 180,E1 8864.892,E2 8864.892} C_VEL
LIN {X 0,Y 615.046,Z 999.418,A -85,B 0,C 180,E1 8867.079,E2 8867.079} C_VEL
LIN {X 0,Y 611.443,Z 1031.876,A -85,B 0,C 180,E1 8868.529,E2 8868.529} C_VEL
LIN {X 0,Y 600.805,Z 1063.275,A -85,B 0,C 180,E1 8869.729,E2 8869.729} C_VEL
LIN {X 0,Y 590.537,Z 1129.8,A -85,B 0,C 180,E1 8874.703,E2 8874.703} C_VEL
LIN {X 0,Y 581.483,Z 1186.553,A -85,B 0,C 180,E1 8880.875,E2 8880.875} C_VEL
LIN {X 0,Y 575.366,Z 1232.589,A -85,B 0,C 180,E1 8888.142,E2 8888.142} C_VEL
LIN {X 0,Y 572.203,Z 1264.521,A -85,B 0,C 180,E1 8895.809,E2 8895.809} C_VEL
LIN {X 0,Y 571.073,Z 1281.721,A -85,B 0,C 180,E1 8903.137,E2 8903.137} C_VEL
LIN {X 0,Y 570.745,Z 1286.838,A -85,B 0,C 180,E1 8909.239,E2 8909.239} C_VEL
LIN {X 0,Y 570.931,Z 1282.883,A -85,B 0,C 180,E1 8916.099,E2 8916.099} C_VEL
LIN {X 0,Y 571.552,Z 1267.995,A -85,B 0,C 180,E1 8923.034,E2 8923.034} C_VEL
LIN {X 0,Y 574.214,Z 1239.99,A -85,B 0,C 180,E1 8930.372,E2 8930.372} C_VEL
LIN {X 0,Y 579.863,Z 1197.292,A -85,B 0,C 180,E1 8937.66,E2 8937.66} C_VEL
LIN {X 0,Y 588.439,Z 1142.215,A -85,B 0,C 180,E1 8944.127,E2 8944.127} C_VEL
LIN {X 0,Y 598.693,Z 1077.626,A -85,B 0,C 180,E1 8949.351,E2 8949.351} C_VEL
LIN {X 0,Y 608.39,Z 1007.206,A -85,B 0,C 180,E1 8953.111,E2 8953.111} C_VEL
LIN {X 0,Y 615.097,Z 938.315,A -85,B 0,C 180,E1 8955.338,E2 8955.338} C_VEL
LIN {X 0,Y 614.819,Z 918.699,A -85,B 0,C 180,E1 8955.903,E2 8955.903} C_VEL
LIN {X 0,Y 571.869,Z 848.798,A -85,B 0,C 180,E1 8962.046,E2 8962.046} C_VEL
LIN {X 0,Y 570.293,Z 844.06,A -85,B 0,C 180,E1 8962.504,E2 8962.504} C_VEL
LIN {X 0,Y 570.216,Z 844.06,A -85,B 0,C 180,E1 8970.544,E2 8970.544} C_VEL
LIN {X 0,Y 570.26,Z 844.06,A -85,B 0,C 180,E1 8980.604,E2 8980.604} C_VEL
LIN {X 0,Y 570.631,Z 844.06,A -85,B 0,C 180,E1 8990.074,E2 8990.074} C_VEL
LIN {X 0,Y 571.206,Z 844.06,A -85,B 0,C 180,E1 8997.742,E2 8997.742} C_VEL
LIN {X 0,Y 570.563,Z 844.06,A -85,B 0,C 180,E1 9006.897,E2 9006.897} C_VEL
LIN {X 0,Y 570.354,Z 844.06,A -85,B 0,C 180,E1 9014.662,E2 9014.662} C_VEL
LIN {X 0,Y 569.944,Z 844.06,A -85,B 0,C 180,E1 9023.366,E2 9023.366} C_VEL
LIN {X 0,Y 569.937,Z 844.06,A -85,B 0,C 180,E1 9031.297,E2 9031.297} C_VEL
LIN {X 0,Y 569.979,Z 845.778,A -85,B 0,C 180,E1 9037.759,E2 9037.759} C_VEL
LIN {X 0,Y 609.905,Z 911.122,A -85,B 0,C 180,E1 9043.619,E2 9043.619} C_VEL
LIN {X 0,Y 615.266,Z 926.588,A -85,B 0,C 180,E1 9044.561,E2 9044.561} C_VEL
LIN {X 0,Y 608.457,Z 996.821,A -85,B 0,C 180,E1 9046.816,E2 9046.816} C_VEL
LIN {X 0,Y 598.878,Z 1066.378,A -85,B 0,C 180,E1 9050.523,E2 9050.523} C_VEL
LIN {X 0,Y 588.421,Z 1131.544,A -85,B 0,C 180,E1 9055.756,E2 9055.756} C_VEL
LIN {X 0,Y 579.584,Z 1187.603,A -85,B 0,C 180,E1 9062.326,E2 9062.326} C_VEL
LIN {X 0,Y 574.135,Z 1228.814,A -85,B 0,C 180,E1 9069.337,E2 9069.337} C_VEL
LIN {X 0,Y 571.619,Z 1256.169,A -85,B 0,C 180,E1 9076.303,E2 9076.303} C_VEL
LIN {X 0,Y 571.052,Z 1271.793,A -85,B 0,C 180,E1 9083.136,E2 9083.136} C_VEL
LIN {X 0,Y 571.362,Z 1276.827,A -85,B 0,C 180,E1 9090.76,E2 9090.76} C_VEL
LIN {X 0,Y 571.27,Z 1269.076,A -85,B 0,C 180,E1 9098.396,E2 9098.396} C_VEL
LIN {X 0,Y 572.102,Z 1250.36,A -85,B 0,C 180,E1 9105.372,E2 9105.372} C_VEL
LIN {X 0,Y 575.117,Z 1219.139,A -85,B 0,C 180,E1 9112.48,E2 9112.48} C_VEL
LIN {X 0,Y 581.605,Z 1173.496,A -85,B 0,C 180,E1 9119.482,E2 9119.482} C_VEL
LIN {X 0,Y 591.164,Z 1114.613,A -85,B 0,C 180,E1 9125.717,E2 9125.717} C_VEL
LIN {X 0,Y 601.752,Z 1047.394,A -85,B 0,C 180,E1 9130.558,E2 9130.558} C_VEL
LIN {X 0,Y 610.769,Z 974.168,A -85,B 0,C 180,E1 9133.985,E2 9133.985} C_VEL
LIN {X 0,Y 614.37,Z 920.515,A -85,B 0,C 180,E1 9135.613,E2 9135.613} C_VEL
LIN {X 0,Y 581.795,Z 863.346,A -85,B 0,C 180,E1 9140.333,E2 9140.333} C_VEL
LIN {X 0,Y 569.983,Z 844.06,A -85,B 0,C 180,E1 9142.352,E2 9142.352} C_VEL
LIN {X 0,Y 570.133,Z 844.06,A -85,B 0,C 180,E1 9150.483,E2 9150.483} C_VEL
LIN {X 0,Y 570.319,Z 844.06,A -85,B 0,C 180,E1 9158.929,E2 9158.929} C_VEL
LIN {X 0,Y 571.202,Z 844.06,A -85,B 0,C 180,E1 9168.485,E2 9168.485} C_VEL
LIN {X 0,Y 571.236,Z 844.06,A -85,B 0,C 180,E1 9177.692,E2 9177.692} C_VEL
LIN {X 0,Y 570.561,Z 844.06,A -85,B 0,C 180,E1 9186.847,E2 9186.847} C_VEL
LIN {X 0,Y 570.362,Z 844.06,A -85,B 0,C 180,E1 9194.61,E2 9194.61} C_VEL
LIN {X 0,Y 569.976,Z 844.06,A -85,B 0,C 180,E1 9203.373,E2 9203.373} C_VEL
LIN {X 0,Y 569.983,Z 844.06,A -85,B 0,C 180,E1 9211.236,E2 9211.236} C_VEL
LIN {X 0,Y 569.975,Z 845.844,A -85,B 0,C 180,E1 9217.656,E2 9217.656} C_VEL
LIN {X 0,Y 611.05,Z 912.641,A -85,B 0,C 180,E1 9223.576,E2 9223.576} C_VEL
LIN {X 0,Y 615.889,Z 927.49,A -85,B 0,C 180,E1 9224.424,E2 9224.424} C_VEL
LIN {X 0,Y 608.776,Z 1002.406,A -85,B 0,C 180,E1 9226.682,E2 9226.682} C_VEL
LIN {X 0,Y 600.805,Z 1063.275,A -85,B 0,C 180,E1 9229.729,E2 9229.729} C_VEL
LIN {X 0,Y 589.783,Z 1093.193,A -85,B 0,C 180,E1 9231.232,E2 9231.232} C_VEL
LIN {X 0,Y 578.888,Z 1156.955,A -85,B 0,C 180,E1 9236.926,E2 9236.926} C_VEL
LIN {X 0,Y 570.398,Z 1209.759,A -85,B 0,C 180,E1 9243.813,E2 9243.813} C_VEL
LIN {X 0,Y 565.259,Z 1248.401,A -85,B 0,C 180,E1 9251.219,E2 9251.219} C_VEL
LIN {X 0,Y 563.438,Z 1270.292,A -85,B 0,C 180,E1 9257.565,E2 9257.565} C_VEL
LIN {X 0,Y 562.951,Z 1283.785,A -85,B 0,C 180,E1 9264.59,E2 9264.59} C_VEL
LIN {X 0,Y 562.625,Z 1286.837,A -85,B 0,C 180,E1 9270.772,E2 9270.772} C_VEL
LIN {X 0,Y 563.227,Z 1280.507,A -85,B 0,C 180,E1 9277.737,E2 9277.737} C_VEL
LIN {X 0,Y 564.75,Z 1260.515,A -85,B 0,C 180,E1 9285.577,E2 9285.577} C_VEL
LIN {X 0,Y 568.21,Z 1226.06,A -85,B 0,C 180,E1 9293.401,E2 9293.401} C_VEL
LIN {X 0,Y 575.211,Z 1179.018,A -85,B 0,C 180,E1 9300.499,E2 9300.499} C_VEL
LIN {X 0,Y 585.334,Z 1119.921,A -85,B 0,C 180,E1 9306.643,E2 9306.643} C_VEL
LIN {X 0,Y 596.171,Z 1052.113,A -85,B 0,C 180,E1 9311.431,E2 9311.431} C_VEL
LIN {X 0,Y 605.55,Z 976.858,A -85,B 0,C 180,E1 9314.815,E2 9314.815} C_VEL
LIN {X 0,Y 609.13,Z 922.297,A -85,B 0,C 180,E1 9316.361,E2 9316.361} C_VEL
LIN {X 0,Y 565.452,Z 850.429,A -85,B 0,C 180,E1 9322.852,E2 9322.852} C_VEL
LIN {X 0,Y 562.286,Z 844.06,A -85,B 0,C 180,E1 9323.613,E2 9323.613} C_VEL
LIN {X 0,Y 562.169,Z 844.06,A -85,B 0,C 180,E1 9331.849,E2 9331.849} C_VEL
LIN {X 0,Y 562.286,Z 844.06,A -85,B 0,C 180,E1 9341.951,E2 9341.951} C_VEL
LIN {X 0,Y 562.43,Z 844.06,A -85,B 0,C 180,E1 9351.494,E2 9351.494} C_VEL
LIN {X 0,Y 562.631,Z 844.06,A -85,B 0,C 180,E1 9359.253,E2 9359.253} C_VEL
LIN {X 0,Y 562.529,Z 844.06,A -85,B 0,C 180,E1 9366.996,E2 9366.996} C_VEL
LIN {X 0,Y 562.297,Z 844.06,A -85,B 0,C 180,E1 9374.877,E2 9374.877} C_VEL
LIN {X 0,Y 561.971,Z 844.06,A -85,B 0,C 180,E1 9383.07,E2 9383.07} C_VEL
LIN {X 0,Y 561.859,Z 844.06,A -85,B 0,C 180,E1 9391.799,E2 9391.799} C_VEL
LIN {X 0,Y 562.004,Z 845.66,A -85,B 0,C 180,E1 9396.692,E2 9396.692} C_VEL
LIN {X 0,Y 603.729,Z 913.462,A -85,B 0,C 180,E1 9403.061,E2 9403.061} C_VEL
LIN {X 0,Y 609.319,Z 930.513,A -85,B 0,C 180,E1 9404.116,E2 9404.116} C_VEL
LIN {X 0,Y 601.964,Z 1001.649,A -85,B 0,C 180,E1 9406.485,E2 9406.485} C_VEL
LIN {X 0,Y 591.728,Z 1071.723,A -85,B 0,C 180,E1 9410.366,E2 9410.366} C_VEL
LIN {X 0,Y 580.602,Z 1137.055,A -85,B 0,C 180,E1 9415.835,E2 9415.835} C_VEL
LIN {X 0,Y 571.451,Z 1191.732,A -85,B 0,C 180,E1 9422.534,E2 9422.534} C_VEL
LIN {X 0,Y 566.038,Z 1231.487,A -85,B 0,C 180,E1 9429.592,E2 9429.592} C_VEL
LIN {X 0,Y 563.56,Z 1258.125,A -85,B 0,C 180,E1 9436.777,E2 9436.777} C_VEL
LIN {X 0,Y 563.144,Z 1272.938,A -85,B 0,C 180,E1 9443.816,E2 9443.816} C_VEL
LIN {X 0,Y 563.358,Z 1276.827,A -85,B 0,C 180,E1 9450.771,E2 9450.771} C_VEL
LIN {X 0,Y 563.251,Z 1269.077,A -85,B 0,C 180,E1 9458.516,E2 9458.516} C_VEL
LIN {X 0,Y 564.17,Z 1250.362,A -85,B 0,C 180,E1 9465.593,E2 9465.593} C_VEL
LIN {X 0,Y 567.441,Z 1219.141,A -85,B 0,C 180,E1 9472.801,E2 9472.801} C_VEL
LIN {X 0,Y 574.354,Z 1173.493,A -85,B 0,C 180,E1 9479.893,E2 9479.893} C_VEL
LIN {X 0,Y 584.264,Z 1115.616,A -85,B 0,C 180,E1 9486.106,E2 9486.106} C_VEL
LIN {X 0,Y 595.459,Z 1048.073,A -85,B 0,C 180,E1 9491.037,E2 9491.037} C_VEL
LIN {X 0,Y 605.011,Z 974.172,A -85,B 0,C 180,E1 9494.518,E2 9494.518} C_VEL
LIN {X 0,Y 608.558,Z 923.879,A -85,B 0,C 180,E1 9496.085,E2 9496.085} C_VEL
LIN {X 0,Y 577.578,Z 869.071,A -85,B 0,C 180,E1 9500.732,E2 9500.732} C_VEL
LIN {X 0,Y 561.996,Z 844.06,A -85,B 0,C 180,E1 9503.388,E2 9503.388} C_VEL
LIN {X 0,Y 562.1,Z 844.06,A -85,B 0,C 180,E1 9511.788,E2 9511.788} C_VEL
LIN {X 0,Y 562.255,Z 844.06,A -85,B 0,C 180,E1 9520.263,E2 9520.263} C_VEL
LIN {X 0,Y 563.007,Z 844.06,A -85,B 0,C 180,E1 9529.476,E2 9529.476} C_VEL
LIN {X 0,Y 563.227,Z 844.06,A -85,B 0,C 180,E1 9537.659,E2 9537.659} C_VEL
LIN {X 0,Y 562.53,Z 844.06,A -85,B 0,C 180,E1 9546.945,E2 9546.945} C_VEL
LIN {X 0,Y 562.305,Z 844.06,A -85,B 0,C 180,E1 9554.825,E2 9554.825} C_VEL
LIN {X 0,Y 562.043,Z 844.06,A -85,B 0,C 180,E1 9563.013,E2 9563.013} C_VEL
LIN {X 0,Y 561.903,Z 844.06,A -85,B 0,C 180,E1 9571.77,E2 9571.77} C_VEL
LIN {X 0,Y 561.949,Z 845.553,A -85,B 0,C 180,E1 9576.58,E2 9576.58} C_VEL
LIN {X 0,Y 604.853,Z 915.031,A -85,B 0,C 180,E1 9583.021,E2 9583.021} C_VEL
LIN {X 0,Y 610.195,Z 929.357,A -85,B 0,C 180,E1 9583.927,E2 9583.927} C_VEL
LIN {X 0,Y 602.691,Z 1003.855,A -85,B 0,C 180,E1 9586.213,E2 9586.213} C_VEL
LIN {X 0,Y 592.455,Z 1076.186,A -85,B 0,C 180,E1 9590.043,E2 9590.043} C_VEL
LIN {X 0,Y 589.783,Z 1093.193,A -85,B 0,C 180,E1 9591.232,E2 9591.232} C_VEL
LIN {X 0,Y 578.36,Z 1121.521,A -85,B 0,C 180,E1 9593.005,E2 9593.005} C_VEL
LIN {X 0,Y 567.675,Z 1180.617,A -85,B 0,C 180,E1 9599.275,E2 9599.275} C_VEL
LIN {X 0,Y 560.35,Z 1227.201,A -85,B 0,C 180,E1 9606.472,E2 9606.472} C_VEL
LIN {X 0,Y 556.701,Z 1261.851,A -85,B 0,C 180,E1 9614.597,E2 9614.597} C_VEL
LIN {X 0,Y 555.371,Z 1280.503,A -85,B 0,C 180,E1 9622.153,E2 9622.153} C_VEL
LIN {X 0,Y 554.748,Z 1286.837,A -85,B 0,C 180,E1 9629.217,E2 9629.217} C_VEL
LIN {X 0,Y 554.954,Z 1282.883,A -85,B 0,C 180,E1 9636.275,E2 9636.275} C_VEL
LIN {X 0,Y 555.717,Z 1267.994,A -85,B 0,C 180,E1 9643.413,E2 9643.413} C_VEL
LIN {X 0,Y 558.977,Z 1238.864,A -85,B 0,C 180,E1 9651.192,E2 9651.192} C_VEL
LIN {X 0,Y 565.552,Z 1194.875,A -85,B 0,C 180,E1 9658.784,E2 9658.784} C_VEL
LIN {X 0,Y 575.11,Z 1139.628,A -85,B 0,C 180,E1 9665.315,E2 9665.315} C_VEL
LIN {X 0,Y 586.55,Z 1073.624,A -85,B 0,C 180,E1 9670.637,E2 9670.637} C_VEL
LIN {X 0,Y 597.395,Z 999.824,A -85,B 0,C 180,E1 9674.481,E2 9674.481} C_VEL
LIN {X 0,Y 603.357,Z 925.673,A -85,B 0,C 180,E1 9676.846,E2 9676.846} C_VEL
LIN {X 0,Y 562.025,Z 857.016,A -85,B 0,C 180,E1 9683.177,E2 9683.177} C_VEL
LIN {X 0,Y 554.261,Z 844.06,A -85,B 0,C 180,E1 9684.775,E2 9684.775} C_VEL
LIN {X 0,Y 554.101,Z 844.06,A -85,B 0,C 180,E1 9693.173,E2 9693.173} C_VEL
LIN {X 0,Y 554.238,Z 844.06,A -85,B 0,C 180,E1 9701.68,E2 9701.68} C_VEL
LIN {X 0,Y 554.453,Z 844.06,A -85,B 0,C 180,E1 9711.371,E2 9711.371} C_VEL
LIN {X 0,Y 554.632,Z 844.06,A -85,B 0,C 180,E1 9719.242,E2 9719.242} C_VEL
LIN {X 0,Y 554.527,Z 844.06,A -85,B 0,C 180,E1 9727.097,E2 9727.097} C_VEL
LIN {X 0,Y 554.264,Z 844.06,A -85,B 0,C 180,E1 9735.097,E2 9735.097} C_VEL
LIN {X 0,Y 553.934,Z 844.06,A -85,B 0,C 180,E1 9743.487,E2 9743.487} C_VEL
LIN {X 0,Y 553.774,Z 844.06,A -85,B 0,C 180,E1 9752.319,E2 9752.319} C_VEL
LIN {X 0,Y 553.962,Z 845.568,A -85,B 0,C 180,E1 9755.556,E2 9755.556} C_VEL
LIN {X 0,Y 596.336,Z 913.551,A -85,B 0,C 180,E1 9762.296,E2 9762.296} C_VEL
LIN {X 0,Y 603.547,Z 933.065,A -85,B 0,C 180,E1 9763.63,E2 9763.63} C_VEL
LIN {X 0,Y 595.802,Z 1003.737,A -85,B 0,C 180,E1 9766.04,E2 9766.04} C_VEL
LIN {X 0,Y 585.182,Z 1072.878,A -85,B 0,C 180,E1 9769.923,E2 9769.923} C_VEL
LIN {X 0,Y 573.7,Z 1137.048,A -85,B 0,C 180,E1 9775.366,E2 9775.366} C_VEL
LIN {X 0,Y 564.079,Z 1191.611,A -85,B 0,C 180,E1 9782.125,E2 9782.125} C_VEL
LIN {X 0,Y 558.1,Z 1232.758,A -85,B 0,C 180,E1 9789.587,E2 9789.587} C_VEL
LIN {X 0,Y 555.602,Z 1258.123,A -85,B 0,C 180,E1 9796.585,E2 9796.585} C_VEL
LIN {X 0,Y 555.138,Z 1272.938,A -85,B 0,C 180,E1 9803.727,E2 9803.727} C_VEL
LIN {X 0,Y 555.355,Z 1276.827,A -85,B 0,C 180,E1 9810.782,E2 9810.782} C_VEL
LIN {X 0,Y 555.238,Z 1269.078,A -85,B 0,C 180,E1 9818.64,E2 9818.64} C_VEL
LIN {X 0,Y 556.236,Z 1250.363,A -85,B 0,C 180,E1 9825.822,E2 9825.822} C_VEL
LIN {X 0,Y 559.775,Z 1219.143,A -85,B 0,C 180,E1 9833.131,E2 9833.131} C_VEL
LIN {X 0,Y 567.091,Z 1173.496,A -85,B 0,C 180,E1 9840.316,E2 9840.316} C_VEL
LIN {X 0,Y 577.697,Z 1114.758,A -85,B 0,C 180,E1 9846.67,E2 9846.67} C_VEL
LIN {X 0,Y 589.473,Z 1047.09,A -85,B 0,C 180,E1 9851.624,E2 9851.624} C_VEL
LIN {X 0,Y 599.345,Z 973.854,A -85,B 0,C 180,E1 9855.072,E2 9855.072} C_VEL
LIN {X 0,Y 602.685,Z 926.93,A -85,B 0,C 180,E1 9856.57,E2 9856.57} C_VEL
LIN {X 0,Y 572.865,Z 874.035,A -85,B 0,C 180,E1 9861.216,E2 9861.216} C_VEL
LIN {X 0,Y 553.951,Z 844.06,A -85,B 0,C 180,E1 9864.596,E2 9864.596} C_VEL
LIN {X 0,Y 554.062,Z 844.06,A -85,B 0,C 180,E1 9873.114,E2 9873.114} C_VEL
LIN {X 0,Y 554.272,Z 844.06,A -85,B 0,C 180,E1 9881.627,E2 9881.627} C_VEL
LIN {X 0,Y 554.991,Z 844.06,A -85,B 0,C 180,E1 9889.74,E2 9889.74} C_VEL
LIN {X 0,Y 554.642,Z 844.06,A -85,B 0,C 180,E1 9899.191,E2 9899.191} C_VEL
LIN {X 0,Y 554.525,Z 844.06,A -85,B 0,C 180,E1 9907.046,E2 9907.046} C_VEL
LIN {X 0,Y 554.261,Z 844.06,A -85,B 0,C 180,E1 9915.045,E2 9915.045} C_VEL
LIN {X 0,Y 553.952,Z 844.06,A -85,B 0,C 180,E1 9923.492,E2 9923.492} C_VEL
LIN {X 0,Y 553.847,Z 844.06,A -85,B 0,C 180,E1 9932.254,E2 9932.254} C_VEL
LIN {X 0,Y 554.032,Z 845.778,A -85,B 0,C 180,E1 9935.471,E2 9935.471} C_VEL
LIN {X 0,Y 597.966,Z 915.898,A -85,B 0,C 180,E1 9942.336,E2 9942.336} C_VEL
LIN {X 0,Y 604.339,Z 933.714,A -85,B 0,C 180,E1 9943.475,E2 9943.475} C_VEL
LIN {X 0,Y 596.412,Z 1007.489,A -85,B 0,C 180,E1 9945.826,E2 9945.826} C_VEL
LIN {X 0,Y 585.482,Z 1080.459,A -85,B 0,C 180,E1 9949.813,E2 9949.813} C_VEL
LIN {X 0,Y 578.36,Z 1121.521,A -85,B 0,C 180,E1 9953.005,E2 9953.005} C_VEL
LIN {X 0,Y 566.755,Z 1148.133,A -85,B 0,C 180,E1 9955.057,E2 9955.057} C_VEL
LIN {X 0,Y 557.042,Z 1201.679,A -85,B 0,C 180,E1 9961.799,E2 9961.799} C_VEL
LIN {X 0,Y 550.482,Z 1243.551,A -85,B 0,C 180,E1 9969.526,E2 9969.526} C_VEL
LIN {X 0,Y 547.59,Z 1270.29,A -85,B 0,C 180,E1 9977.199,E2 9977.199} C_VEL
LIN {X 0,Y 546.951,Z 1283.779,A -85,B 0,C 180,E1 9984.431,E2 9984.431} C_VEL
LIN {X 0,Y 546.641,Z 1286.837,A -85,B 0,C 180,E1 9990.795,E2 9990.795} C_VEL
LIN {X 0,Y 547.303,Z 1280.501,A -85,B 0,C 180,E1 9997.964,E2 9997.964} C_VEL
LIN {X 0,Y 548.895,Z 1260.513,A -85,B 0,C 180,E1 10006.039,E2 10006.039} C_VEL
LIN {X 0,Y 552.793,Z 1226.108,A -85,B 0,C 180,E1 10014.084,E2 10014.084} C_VEL
LIN {X 0,Y 560.554,Z 1179.853,A -85,B 0,C 180,E1 10021.267,E2 10021.267} C_VEL
LIN {X 0,Y 571.746,Z 1121.372,A -85,B 0,C 180,E1 10027.508,E2 10027.508} C_VEL
LIN {X 0,Y 583.548,Z 1054.265,A -85,B 0,C 180,E1 10032.363,E2 10032.363} C_VEL
LIN {X 0,Y 593.856,Z 979.088,A -85,B 0,C 180,E1 10035.835,E2 10035.835} C_VEL
LIN {X 0,Y 597.57,Z 929.041,A -85,B 0,C 180,E1 10037.347,E2 10037.347} C_VEL
LIN {X 0,Y 558.169,Z 863.084,A -85,B 0,C 180,E1 10043.579,E2 10043.579} C_VEL
LIN {X 0,Y 546.24,Z 844.06,A -85,B 0,C 180,E1 10046.015,E2 10046.015} C_VEL
LIN {X 0,Y 546.007,Z 844.06,A -85,B 0,C 180,E1 10054.52,E2 10054.52} C_VEL
LIN {X 0,Y 546.199,Z 844.06,A -85,B 0,C 180,E1 10063.315,E2 10063.315} C_VEL
LIN {X 0,Y 546.451,Z 844.06,A -85,B 0,C 180,E1 10071.243,E2 10071.243} C_VEL
LIN {X 0,Y 546.647,Z 844.06,A -85,B 0,C 180,E1 10079.231,E2 10079.231} C_VEL
LIN {X 0,Y 546.495,Z 844.06,A -85,B 0,C 180,E1 10087.202,E2 10087.202} C_VEL
LIN {X 0,Y 546.216,Z 844.06,A -85,B 0,C 180,E1 10095.325,E2 10095.325} C_VEL
LIN {X 0,Y 545.91,Z 844.06,A -85,B 0,C 180,E1 10103.79,E2 10103.79} C_VEL
LIN {X 0,Y 545.758,Z 844.06,A -85,B 0,C 180,E1 10112.853,E2 10112.853} C_VEL
LIN {X 0,Y 545.982,Z 845.992,A -85,B 0,C 180,E1 10114.375,E2 10114.375} C_VEL
LIN {X 0,Y 586.82,Z 909.627,A -85,B 0,C 180,E1 10121.149,E2 10121.149} C_VEL
LIN {X 0,Y 597.778,Z 935.979,A -85,B 0,C 180,E1 10123.143,E2 10123.143} C_VEL
LIN {X 0,Y 589.628,Z 1006.293,A -85,B 0,C 180,E1 10125.608,E2 10125.608} C_VEL
LIN {X 0,Y 578.342,Z 1075.859,A -85,B 0,C 180,E1 10129.608,E2 10129.608} C_VEL
LIN {X 0,Y 566.05,Z 1140.886,A -85,B 0,C 180,E1 10135.297,E2 10135.297} C_VEL
LIN {X 0,Y 556.008,Z 1195.238,A -85,B 0,C 180,E1 10142.289,E2 10142.289} C_VEL
LIN {X 0,Y 550.232,Z 1233.589,A -85,B 0,C 180,E1 10149.481,E2 10149.481} C_VEL
LIN {X 0,Y 547.608,Z 1259.269,A -85,B 0,C 180,E1 10156.793,E2 10156.793} C_VEL
LIN {X 0,Y 547.273,Z 1273.829,A -85,B 0,C 180,E1 10164.434,E2 10164.434} C_VEL
LIN {X 0,Y 547.212,Z 1276.352,A -85,B 0,C 180,E1 10172.383,E2 10172.383} C_VEL
LIN {X 0,Y 547.216,Z 1267.802,A -85,B 0,C 180,E1 10179.425,E2 10179.425} C_VEL
LIN {X 0,Y 548.45,Z 1249.02,A -85,B 0,C 180,E1 10186.465,E2 10186.465} C_VEL
LIN {X 0,Y 552.484,Z 1216.971,A -85,B 0,C 180,E1 10193.884,E2 10193.884} C_VEL
LIN {X 0,Y 560.402,Z 1170.193,A -85,B 0,C 180,E1 10201.183,E2 10201.183} C_VEL
LIN {X 0,Y 571.848,Z 1110.579,A -85,B 0,C 180,E1 10207.545,E2 10207.545} C_VEL
LIN {X 0,Y 583.824,Z 1044.44,A -85,B 0,C 180,E1 10212.322,E2 10212.322} C_VEL
LIN {X 0,Y 594.014,Z 971.464,A -85,B 0,C 180,E1 10215.707,E2 10215.707} C_VEL
LIN {X 0,Y 596.82,Z 930.067,A -85,B 0,C 180,E1 10217.066,E2 10217.066} C_VEL
LIN {X 0,Y 567.301,Z 877.308,A -85,B 0,C 180,E1 10221.858,E2 10221.858} C_VEL
LIN {X 0,Y 545.948,Z 844.06,A -85,B 0,C 180,E1 10225.653,E2 10225.653} C_VEL
LIN {X 0,Y 546.097,Z 844.06,A -85,B 0,C 180,E1 10234.494,E2 10234.494} C_VEL
LIN {X 0,Y 546.49,Z 844.06,A -85,B 0,C 180,E1 10243.215,E2 10243.215} C_VEL
LIN {X 0,Y 546.655,Z 844.06,A -85,B 0,C 180,E1 10251.194,E2 10251.194} C_VEL
LIN {X 0,Y 546.657,Z 844.06,A -85,B 0,C 180,E1 10259.179,E2 10259.179} C_VEL
LIN {X 0,Y 546.497,Z 844.06,A -85,B 0,C 180,E1 10267.15,E2 10267.15} C_VEL
LIN {X 0,Y 546.211,Z 844.06,A -85,B 0,C 180,E1 10275.272,E2 10275.272} C_VEL
LIN {X 0,Y 545.929,Z 844.06,A -85,B 0,C 180,E1 10283.733,E2 10283.733} C_VEL
LIN {X 0,Y 545.821,Z 844.06,A -85,B 0,C 180,E1 10292.787,E2 10292.787} C_VEL
LIN {X 0,Y 546.059,Z 846.129,A -85,B 0,C 180,E1 10294.291,E2 10294.291} C_VEL
LIN {X 0,Y 587.877,Z 910.992,A -85,B 0,C 180,E1 10301.118,E2 10301.118} C_VEL
LIN {X 0,Y 598.625,Z 935.961,A -85,B 0,C 180,E1 10302.973,E2 10302.973} C_VEL
LIN {X 0,Y 590.313,Z 1009.696,A -85,B 0,C 180,E1 10305.37,E2 10305.37} C_VEL
LIN {X 0,Y 578.908,Z 1081.957,A -85,B 0,C 180,E1 10309.39,E2 10309.39} C_VEL
LIN {X 0,Y 567.062,Z 1146.671,A -85,B 0,C 180,E1 10314.901,E2 10314.901} C_VEL
LIN {X 0,Y 566.755,Z 1148.133,A -85,B 0,C 180,E1 10315.057,E2 10315.057} C_VEL
LIN {X 0,Y 554.796,Z 1172.76,A -85,B 0,C 180,E1 10317.368,E2 10317.368} C_VEL
LIN {X 0,Y 545.84,Z 1221.269,A -85,B 0,C 180,E1 10324.634,E2 10324.634} C_VEL
LIN {X 0,Y 541.127,Z 1254.88,A -85,B 0,C 180,E1 10332.079,E2 10332.079} C_VEL
LIN {X 0,Y 539.403,Z 1276.028,A -85,B 0,C 180,E1 10339.47,E2 10339.47} C_VEL
LIN {X 0,Y 539.286,Z 1286.381,A -85,B 0,C 180,E1 10347.582,E2 10347.582} C_VEL
LIN {X 0,Y 539.019,Z 1283.778,A -85,B 0,C 180,E1 10355.651,E2 10355.651} C_VEL
LIN {X 0,Y 539.642,Z 1270.291,A -85,B 0,C 180,E1 10362.992,E2 10362.992} C_VEL
LIN {X 0,Y 542.758,Z 1243.35,A -85,B 0,C 180,E1 10370.827,E2 10370.827} C_VEL
LIN {X 0,Y 549.953,Z 1200.158,A -85,B 0,C 180,E1 10378.854,E2 10378.854} C_VEL
LIN {X 0,Y 560.47,Z 1145.026,A -85,B 0,C 180,E1 10385.765,E2 10385.765} C_VEL
LIN {X 0,Y 572.986,Z 1079.801,A -85,B 0,C 180,E1 10391.29,E2 10391.29} C_VEL
LIN {X 0,Y 584.826,Z 1008.021,A -85,B 0,C 180,E1 10395.249,E2 10395.249} C_VEL
LIN {X 0,Y 592.883,Z 937.894,A -85,B 0,C 180,E1 10397.556,E2 10397.556} C_VEL
LIN {X 0,Y 565.67,Z 886.282,A -85,B 0,C 180,E1 10402.092,E2 10402.092} C_VEL
LIN {X 0,Y 538.187,Z 844.06,A -85,B 0,C 180,E1 10407.174,E2 10407.174} C_VEL
LIN {X 0,Y 537.919,Z 844.06,A -85,B 0,C 180,E1 10416.385,E2 10416.385} C_VEL
LIN {X 0,Y 538.106,Z 844.06,A -85,B 0,C 180,E1 10424.492,E2 10424.492} C_VEL
LIN {X 0,Y 538.318,Z 844.06,A -85,B 0,C 180,E1 10432.741,E2 10432.741} C_VEL
LIN {X 0,Y 538.65,Z 844.06,A -85,B 0,C 180,E1 10439.219,E2 10439.219} C_VEL
LIN {X 0,Y 538.464,Z 844.06,A -85,B 0,C 180,E1 10447.31,E2 10447.31} C_VEL
LIN {X 0,Y 538.193,Z 844.06,A -85,B 0,C 180,E1 10455.559,E2 10455.559} C_VEL
LIN {X 0,Y 537.88,Z 844.06,A -85,B 0,C 180,E1 10464.168,E2 10464.168} C_VEL
LIN {X 0,Y 537.925,Z 845.693,A -85,B 0,C 180,E1 10473.09,E2 10473.09} C_VEL
LIN {X 0,Y 577.428,Z 906.517,A -85,B 0,C 180,E1 10479.975,E2 10479.975} C_VEL
LIN {X 0,Y 592.077,Z 938.774,A -85,B 0,C 180,E1 10482.645,E2 10482.645} C_VEL
LIN {X 0,Y 583.326,Z 1009.733,A -85,B 0,C 180,E1 10485.206,E2 10485.206} C_VEL
LIN {X 0,Y 571.484,Z 1078.899,A -85,B 0,C 180,E1 10489.289,E2 10489.289} C_VEL
LIN {X 0,Y 558.793,Z 1142.811,A -85,B 0,C 180,E1 10495.019,E2 10495.019} C_VEL
LIN {X 0,Y 548.571,Z 1195.441,A -85,B 0,C 180,E1 10501.916,E2 10501.916} C_VEL
LIN {X 0,Y 542.526,Z 1233.357,A -85,B 0,C 180,E1 10509.121,E2 10509.121} C_VEL
LIN {X 0,Y 539.726,Z 1258.118,A -85,B 0,C 180,E1 10516.182,E2 10516.182} C_VEL
LIN {X 0,Y 539.138,Z 1272.936,A -85,B 0,C 180,E1 10523.54,E2 10523.54} C_VEL
LIN {X 0,Y 539.374,Z 1276.827,A -85,B 0,C 180,E1 10530.806,E2 10530.806} C_VEL
LIN {X 0,Y 539.375,Z 1270.431,A -85,B 0,C 180,E1 10538.082,E2 10538.082} C_VEL
LIN {X 0,Y 540.355,Z 1251.705,A -85,B 0,C 180,E1 10545.881,E2 10545.881} C_VEL
LIN {X 0,Y 544.247,Z 1220.876,A -85,B 0,C 180,E1 10553.484,E2 10553.484} C_VEL
LIN {X 0,Y 552.221,Z 1175.889,A -85,B 0,C 180,E1 10560.88,E2 10560.88} C_VEL
LIN {X 0,Y 563.883,Z 1117.637,A -85,B 0,C 180,E1 10567.431,E2 10567.431} C_VEL
LIN {X 0,Y 576.561,Z 1051.697,A -85,B 0,C 180,E1 10572.443,E2 10572.443} C_VEL
LIN {X 0,Y 587.436,Z 978.707,A -85,B 0,C 180,E1 10576.028,E2 10576.028} C_VEL
LIN {X 0,Y 591.146,Z 933.553,A -85,B 0,C 180,E1 10577.544,E2 10577.544} C_VEL
LIN {X 0,Y 561.617,Z 880.453,A -85,B 0,C 180,E1 10582.54,E2 10582.54} C_VEL
LIN {X 0,Y 537.982,Z 844.06,A -85,B 0,C 180,E1 10586.988,E2 10586.988} C_VEL
LIN {X 0,Y 538.199,Z 844.06,A -85,B 0,C 180,E1 10596.317,E2 10596.317} C_VEL
LIN {X 0,Y 538.971,Z 844.06,A -85,B 0,C 180,E1 10606.131,E2 10606.131} C_VEL
LIN {X 0,Y 539.058,Z 844.06,A -85,B 0,C 180,E1 10616.77,E2 10616.77} C_VEL
LIN {X 0,Y 538.849,Z 844.06,A -85,B 0,C 180,E1 10625.629,E2 10625.629} C_VEL
LIN {X 0,Y 538.182,Z 844.06,A -85,B 0,C 180,E1 10635.505,E2 10635.505} C_VEL
LIN {X 0,Y 537.895,Z 844.06,A -85,B 0,C 180,E1 10644.11,E2 10644.11} C_VEL
LIN {X 0,Y 537.987,Z 845.795,A -85,B 0,C 180,E1 10653.006,E2 10653.006} C_VEL
LIN {X 0,Y 578.088,Z 907.399,A -85,B 0,C 180,E1 10659.918,E2 10659.918} C_VEL
LIN {X 0,Y 592.82,Z 939.469,A -85,B 0,C 180,E1 10662.491,E2 10662.491} C_VEL
LIN {X 0,Y 584.145,Z 1012.163,A -85,B 0,C 180,E1 10664.925,E2 10664.925} C_VEL
LIN {X 0,Y 572.065,Z 1084.716,A -85,B 0,C 180,E1 10669.056,E2 10669.056} C_VEL
LIN {X 0,Y 559.832,Z 1148.587,A -85,B 0,C 180,E1 10674.618,E2 10674.618} C_VEL
LIN {X 0,Y 554.796,Z 1172.76,A -85,B 0,C 180,E1 10677.368,E2 10677.368} C_VEL
LIN {X 0,Y 543.438,Z 1195.214,A -85,B 0,C 180,E1 10679.982,E2 10679.982} C_VEL
LIN {X 0,Y 535.823,Z 1239.446,A -85,B 0,C 180,E1 10687.975,E2 10687.975} C_VEL
LIN {X 0,Y 531.93,Z 1269.14,A -85,B 0,C 180,E1 10696.396,E2 10696.396} C_VEL
LIN {X 0,Y 531.081,Z 1282.881,A -85,B 0,C 180,E1 10703.441,E2 10703.441} C_VEL
LIN {X 0,Y 530.776,Z 1286.837,A -85,B 0,C 180,E1 10709.181,E2 10709.181} C_VEL
LIN {X 0,Y 531.039,Z 1282.882,A -85,B 0,C 180,E1 10716.559,E2 10716.559} C_VEL
LIN {X 0,Y 532.386,Z 1266.143,A -85,B 0,C 180,E1 10724.69,E2 10724.69} C_VEL
LIN {X 0,Y 536.345,Z 1235.515,A -85,B 0,C 180,E1 10732.884,E2 10732.884} C_VEL
LIN {X 0,Y 544.242,Z 1191.046,A -85,B 0,C 180,E1 10740.629,E2 10740.629} C_VEL
LIN {X 0,Y 555.75,Z 1135.002,A -85,B 0,C 180,E1 10747.261,E2 10747.261} C_VEL
LIN {X 0,Y 568.679,Z 1068.759,A -85,B 0,C 180,E1 10752.586,E2 10752.586} C_VEL
LIN {X 0,Y 580.848,Z 994.727,A -85,B 0,C 180,E1 10756.375,E2 10756.375} C_VEL
LIN {X 0,Y 586.29,Z 936.36,A -85,B 0,C 180,E1 10758.316,E2 10758.316} C_VEL
LIN {X 0,Y 550.135,Z 874.399,A -85,B 0,C 180,E1 10764.477,E2 10764.477} C_VEL
LIN {X 0,Y 530.112,Z 844.06,A -85,B 0,C 180,E1 10768.409,E2 10768.409} C_VEL
LIN {X 0,Y 529.891,Z 844.06,A -85,B 0,C 180,E1 10777.292,E2 10777.292} C_VEL
LIN {X 0,Y 530.138,Z 844.06,A -85,B 0,C 180,E1 10785.95,E2 10785.95} C_VEL
LIN {X 0,Y 530.943,Z 844.06,A -85,B 0,C 180,E1 10795.93,E2 10795.93} C_VEL
LIN {X 0,Y 530.819,Z 844.06,A -85,B 0,C 180,E1 10805.767,E2 10805.767} C_VEL
LIN {X 0,Y 530.146,Z 844.06,A -85,B 0,C 180,E1 10815.802,E2 10815.802} C_VEL
LIN {X 0,Y 529.821,Z 844.06,A -85,B 0,C 180,E1 10824.56,E2 10824.56} C_VEL
LIN {X 0,Y 529.975,Z 845.877,A -85,B 0,C 180,E1 10831.748,E2 10831.748} C_VEL
LIN {X 0,Y 566.981,Z 901.721,A -85,B 0,C 180,E1 10838.561,E2 10838.561} C_VEL
LIN {X 0,Y 586.499,Z 940.381,A -85,B 0,C 180,E1 10842.103,E2 10842.103} C_VEL
LIN {X 0,Y 577.218,Z 1012.182,A -85,B 0,C 180,E1 10844.749,E2 10844.749} C_VEL
LIN {X 0,Y 564.886,Z 1080.737,A -85,B 0,C 180,E1 10848.872,E2 10848.872} C_VEL
LIN {X 0,Y 551.714,Z 1144.051,A -85,B 0,C 180,E1 10854.65,E2 10854.65} C_VEL
LIN {X 0,Y 540.911,Z 1196.923,A -85,B 0,C 180,E1 10861.738,E2 10861.738} C_VEL
LIN {X 0,Y 534.511,Z 1235.093,A -85,B 0,C 180,E1 10869.228,E2 10869.228} C_VEL
LIN {X 0,Y 531.675,Z 1260.41,A -85,B 0,C 180,E1 10876.81,E2 10876.81} C_VEL
LIN {X 0,Y 531.241,Z 1273.822,A -85,B 0,C 180,E1 10884.266,E2 10884.266} C_VEL
LIN {X 0,Y 531.223,Z 1276.353,A -85,B 0,C 180,E1 10892.454,E2 10892.454} C_VEL
LIN {X 0,Y 531.277,Z 1267.745,A -85,B 0,C 180,E1 10899.738,E2 10899.738} C_VEL
LIN {X 0,Y 532.67,Z 1249.027,A -85,B 0,C 180,E1 10906.967,E2 10906.967} C_VEL
LIN {X 0,Y 537.161,Z 1217.32,A -85,B 0,C 180,E1 10914.539,E2 10914.539} C_VEL
LIN {X 0,Y 546.055,Z 1170.681,A -85,B 0,C 180,E1 10922.028,E2 10922.028} C_VEL
LIN {X 0,Y 558.558,Z 1111.531,A -85,B 0,C 180,E1 10928.519,E2 10928.519} C_VEL
LIN {X 0,Y 571.858,Z 1044.179,A -85,B 0,C 180,E1 10933.459,E2 10933.459} C_VEL
LIN {X 0,Y 582.637,Z 973.323,A -85,B 0,C 180,E1 10936.786,E2 10936.786} C_VEL
LIN {X 0,Y 585.48,Z 936.997,A -85,B 0,C 180,E1 10938.036,E2 10938.036} C_VEL
LIN {X 0,Y 555.183,Z 882.156,A -85,B 0,C 180,E1 10943.383,E2 10943.383} C_VEL
LIN {X 0,Y 530.012,Z 844.06,A -85,B 0,C 180,E1 10948.386,E2 10948.386} C_VEL
LIN {X 0,Y 530.191,Z 844.06,A -85,B 0,C 180,E1 10958.375,E2 10958.375} C_VEL
LIN {X 0,Y 531.08,Z 844.06,A -85,B 0,C 180,E1 10967.602,E2 10967.602} C_VEL
LIN {X 0,Y 531.212,Z 844.06,A -85,B 0,C 180,E1 10977.518,E2 10977.518} C_VEL
LIN {X 0,Y 530.445,Z 844.06,A -85,B 0,C 180,E1 10987.367,E2 10987.367} C_VEL
LIN {X 0,Y 530.084,Z 844.06,A -85,B 0,C 180,E1 10996.582,E2 10996.582} C_VEL
LIN {X 0,Y 529.819,Z 844.06,A -85,B 0,C 180,E1 11005.625,E2 11005.625} C_VEL
LIN {X 0,Y 530.02,Z 845.779,A -85,B 0,C 180,E1 11011.661,E2 11011.661} C_VEL
LIN {X 0,Y 567.765,Z 902.989,A -85,B 0,C 180,E1 11018.557,E2 11018.557} C_VEL
LIN {X 0,Y 587.206,Z 941.383,A -85,B 0,C 180,E1 11021.96,E2 11021.96} C_VEL
LIN {X 0,Y 577.985,Z 1014.984,A -85,B 0,C 180,E1 11024.491,E2 11024.491} C_VEL
LIN {X 0,Y 565.314,Z 1087.086,A -85,B 0,C 180,E1 11028.685,E2 11028.685} C_VEL
LIN {X 0,Y 552.544,Z 1150.607,A -85,B 0,C 180,E1 11034.344,E2 11034.344} C_VEL
LIN {X 0,Y 543.438,Z 1195.214,A -85,B 0,C 180,E1 11039.982,E2 11039.982} C_VEL
LIN {X 0,Y 531.971,Z 1215.556,A -85,B 0,C 180,E1 11042.841,E2 11042.841} C_VEL
LIN {X 0,Y 525.845,Z 1251.682,A -85,B 0,C 180,E1 11050.63,E2 11050.63} C_VEL
LIN {X 0,Y 523.399,Z 1274.186,A -85,B 0,C 180,E1 11058.298,E2 11058.298} C_VEL
LIN {X 0,Y 523.242,Z 1285.35,A -85,B 0,C 180,E1 11065.845,E2 11065.845} C_VEL
LIN {X 0,Y 523.263,Z 1285.351,A -85,B 0,C 180,E1 11074.155,E2 11074.155} C_VEL
LIN {X 0,Y 523.474,Z 1274.186,A -85,B 0,C 180,E1 11081.7,E2 11081.7} C_VEL
LIN {X 0,Y 525.829,Z 1251.681,A -85,B 0,C 180,E1 11089.37,E2 11089.37} C_VEL
LIN {X 0,Y 532.076,Z 1214.465,A -85,B 0,C 180,E1 11097.361,E2 11097.361} C_VEL
LIN {X 0,Y 542.815,Z 1163.156,A -85,B 0,C 180,E1 11104.751,E2 11104.751} C_VEL
LIN {X 0,Y 556.412,Z 1100.459,A -85,B 0,C 180,E1 11110.854,E2 11110.854} C_VEL
LIN {X 0,Y 569.635,Z 1031.67,A -85,B 0,C 180,E1 11115.275,E2 11115.275} C_VEL
LIN {X 0,Y 579.801,Z 959.458,A -85,B 0,C 180,E1 11118.157,E2 11118.157} C_VEL
LIN {X 0,Y 580.429,Z 939.714,A -85,B 0,C 180,E1 11118.846,E2 11118.846} C_VEL
LIN {X 0,Y 546.252,Z 880.015,A -85,B 0,C 180,E1 11124.924,E2 11124.924} C_VEL
LIN {X 0,Y 522.109,Z 844.06,A -85,B 0,C 180,E1 11129.873,E2 11129.873} C_VEL
LIN {X 0,Y 521.932,Z 844.06,A -85,B 0,C 180,E1 11138.725,E2 11138.725} C_VEL
LIN {X 0,Y 522.274,Z 844.06,A -85,B 0,C 180,E1 11147.445,E2 11147.445} C_VEL
LIN {X 0,Y 523.184,Z 844.06,A -85,B 0,C 180,E1 11157.534,E2 11157.534} C_VEL
LIN {X 0,Y 522.802,Z 844.06,A -85,B 0,C 180,E1 11165.856,E2 11165.856} C_VEL
LIN {X 0,Y 522.113,Z 844.06,A -85,B 0,C 180,E1 11176.051,E2 11176.051} C_VEL
LIN {X 0,Y 521.789,Z 844.06,A -85,B 0,C 180,E1 11184.963,E2 11184.963} C_VEL
LIN {X 0,Y 522.019,Z 845.956,A -85,B 0,C 180,E1 11190.307,E2 11190.307} C_VEL
LIN {X 0,Y 558.46,Z 899.815,A -85,B 0,C 180,E1 11197.402,E2 11197.402} C_VEL
LIN {X 0,Y 580.702,Z 944.538,A -85,B 0,C 180,E1 11201.621,E2 11201.621} C_VEL
LIN {X 0,Y 571.002,Z 1015.387,A -85,B 0,C 180,E1 11204.316,E2 11204.316} C_VEL
LIN {X 0,Y 558.033,Z 1084.149,A -85,B 0,C 180,E1 11208.567,E2 11208.567} C_VEL
LIN {X 0,Y 544.401,Z 1146.583,A -85,B 0,C 180,E1 11214.417,E2 11214.417} C_VEL
LIN {X 0,Y 532.975,Z 1199.959,A -85,B 0,C 180,E1 11221.809,E2 11221.809} C_VEL
LIN {X 0,Y 526.371,Z 1237.789,A -85,B 0,C 180,E1 11229.576,E2 11229.576} C_VEL
LIN {X 0,Y 523.635,Z 1262.36,A -85,B 0,C 180,E1 11237.455,E2 11237.455} C_VEL
LIN {X 0,Y 523.242,Z 1273.818,A -85,B 0,C 180,E1 11244.178,E2 11244.178} C_VEL
LIN {X 0,Y 523.217,Z 1276.354,A -85,B 0,C 180,E1 11252.492,E2 11252.492} C_VEL
LIN {X 0,Y 523.284,Z 1267.744,A -85,B 0,C 180,E1 11259.889,E2 11259.889} C_VEL
LIN {X 0,Y 525.065,Z 1247.661,A -85,B 0,C 180,E1 11267.654,E2 11267.654} C_VEL
LIN {X 0,Y 530.651,Z 1212.356,A -85,B 0,C 180,E1 11275.892,E2 11275.892} C_VEL
LIN {X 0,Y 541.089,Z 1162.081,A -85,B 0,C 180,E1 11283.625,E2 11283.625} C_VEL
LIN {X 0,Y 554.224,Z 1102.064,A -85,B 0,C 180,E1 11289.899,E2 11289.899} C_VEL
LIN {X 0,Y 567.793,Z 1034.308,A -85,B 0,C 180,E1 11294.604,E2 11294.604} C_VEL
LIN {X 0,Y 578.446,Z 964.525,A -85,B 0,C 180,E1 11297.671,E2 11297.671} C_VEL
LIN {X 0,Y 579.72,Z 940.104,A -85,B 0,C 180,E1 11298.565,E2 11298.565} C_VEL
LIN {X 0,Y 548.373,Z 883.324,A -85,B 0,C 180,E1 11304.329,E2 11304.329} C_VEL
LIN {X 0,Y 521.987,Z 844.06,A -85,B 0,C 180,E1 11309.847,E2 11309.847} C_VEL
LIN {X 0,Y 522.182,Z 844.06,A -85,B 0,C 180,E1 11318.677,E2 11318.677} C_VEL
LIN {X 0,Y 523.039,Z 844.06,A -85,B 0,C 180,E1 11327.408,E2 11327.408} C_VEL
LIN {X 0,Y 523.21,Z 844.06,A -85,B 0,C 180,E1 11337.48,E2 11337.48} C_VEL
LIN {X 0,Y 522.795,Z 844.06,A -85,B 0,C 180,E1 11345.802,E2 11345.802} C_VEL
LIN {X 0,Y 522.336,Z 844.06,A -85,B 0,C 180,E1 11354.264,E2 11354.264} C_VEL
LIN {X 0,Y 521.834,Z 844.06,A -85,B 0,C 180,E1 11363.731,E2 11363.731} C_VEL
LIN {X 0,Y 522.03,Z 845.73,A -85,B 0,C 180,E1 11370.213,E2 11370.213} C_VEL
LIN {X 0,Y 558.719,Z 900.347,A -85,B 0,C 180,E1 11377.318,E2 11377.318} C_VEL
LIN {X 0,Y 581.524,Z 944.871,A -85,B 0,C 180,E1 11381.461,E2 11381.461} C_VEL
LIN {X 0,Y 572.106,Z 1015.932,A -85,B 0,C 180,E1 11383.955,E2 11383.955} C_VEL
LIN {X 0,Y 559.134,Z 1086.944,A -85,B 0,C 180,E1 11388.121,E2 11388.121} C_VEL
LIN {X 0,Y 545.486,Z 1151.656,A -85,B 0,C 180,E1 11393.956,E2 11393.956} C_VEL
LIN {X 0,Y 534.499,Z 1204.149,A -85,B 0,C 180,E1 11400.929,E2 11400.929} C_VEL
LIN {X 0,Y 531.971,Z 1215.556,A -85,B 0,C 180,E1 11402.841,E2 11402.841} C_VEL
LIN {X 0,Y 521.219,Z 1233.551,A -85,B 0,C 180,E1 11405.954,E2 11405.954} C_VEL
LIN {X 0,Y 516.806,Z 1265.691,A -85,B 0,C 180,E1 11414.686,E2 11414.686} C_VEL
LIN {X 0,Y 515.116,Z 1282.881,A -85,B 0,C 180,E1 11423.237,E2 11423.237} C_VEL
LIN {X 0,Y 514.81,Z 1286.837,A -85,B 0,C 180,E1 11429.156,E2 11429.156} C_VEL
LIN {X 0,Y 515.067,Z 1282.882,A -85,B 0,C 180,E1 11436.764,E2 11436.764} C_VEL
LIN {X 0,Y 516.716,Z 1265.693,A -85,B 0,C 180,E1 11445.316,E2 11445.316} C_VEL
LIN {X 0,Y 521.088,Z 1234.872,A -85,B 0,C 180,E1 11453.743,E2 11453.743} C_VEL
LIN {X 0,Y 529.948,Z 1190.224,A -85,B 0,C 180,E1 11461.672,E2 11461.672} C_VEL
LIN {X 0,Y 542.69,Z 1134.035,A -85,B 0,C 180,E1 11468.413,E2 11468.413} C_VEL
LIN {X 0,Y 556.687,Z 1068.465,A -85,B 0,C 180,E1 11473.741,E2 11473.741} C_VEL
LIN {X 0,Y 569.773,Z 993.931,A -85,B 0,C 180,E1 11477.592,E2 11477.592} C_VEL
LIN {X 0,Y 574.972,Z 943.652,A -85,B 0,C 180,E1 11479.325,E2 11479.325} C_VEL
LIN {X 0,Y 542.275,Z 885.398,A -85,B 0,C 180,E1 11485.403,E2 11485.403} C_VEL
LIN {X 0,Y 513.995,Z 844.06,A -85,B 0,C 180,E1 11491.667,E2 11491.667} C_VEL
LIN {X 0,Y 514.092,Z 844.06,A -85,B 0,C 180,E1 11501.979,E2 11501.979} C_VEL
LIN {X 0,Y 514.433,Z 844.06,A -85,B 0,C 180,E1 11510.957,E2 11510.957} C_VEL
LIN {X 0,Y 514.676,Z 844.06,A -85,B 0,C 180,E1 11519.183,E2 11519.183} C_VEL
LIN {X 0,Y 514.405,Z 844.06,A -85,B 0,C 180,E1 11527.654,E2 11527.654} C_VEL
LIN {X 0,Y 514.047,Z 844.06,A -85,B 0,C 180,E1 11536.502,E2 11536.502} C_VEL
LIN {X 0,Y 513.734,Z 844.06,A -85,B 0,C 180,E1 11545.795,E2 11545.795} C_VEL
LIN {X 0,Y 514.015,Z 845.868,A -85,B 0,C 180,E1 11548.738,E2 11548.738} C_VEL
LIN {X 0,Y 549.397,Z 897.401,A -85,B 0,C 180,E1 11556.082,E2 11556.082} C_VEL
LIN {X 0,Y 575.128,Z 946.825,A -85,B 0,C 180,E1 11561.089,E2 11561.089} C_VEL
LIN {X 0,Y 564.777,Z 1018.885,A -85,B 0,C 180,E1 11563.888,E2 11563.888} C_VEL
LIN {X 0,Y 551.159,Z 1087.77,A -85,B 0,C 180,E1 11568.271,E2 11568.271} C_VEL
LIN {X 0,Y 536.861,Z 1150.114,A -85,B 0,C 180,E1 11574.289,E2 11574.289} C_VEL
LIN {X 0,Y 525.012,Z 1202.728,A -85,B 0,C 180,E1 11581.857,E2 11581.857} C_VEL
LIN {X 0,Y 518.328,Z 1239.915,A -85,B 0,C 180,E1 11589.792,E2 11589.792} C_VEL
LIN {X 0,Y 515.669,Z 1264.286,A -85,B 0,C 180,E1 11598.12,E2 11598.12} C_VEL
LIN {X 0,Y 515.197,Z 1275.378,A -85,B 0,C 180,E1 11605.78,E2 11605.78} C_VEL
LIN {X 0,Y 515.209,Z 1276.354,A -85,B 0,C 180,E1 11612.531,E2 11612.531} C_VEL
LIN {X 0,Y 515.324,Z 1267.511,A -85,B 0,C 180,E1 11620.169,E2 11620.169} C_VEL
LIN {X 0,Y 517.253,Z 1247.663,A -85,B 0,C 180,E1 11627.93,E2 11627.93} C_VEL
LIN {X 0,Y 523.486,Z 1211.312,A -85,B 0,C 180,E1 11636.478,E2 11636.478} C_VEL
LIN {X 0,Y 534.46,Z 1160.621,A -85,B 0,C 180,E1 11644.318,E2 11644.318} C_VEL
LIN {X 0,Y 548.419,Z 1099.874,A -85,B 0,C 180,E1 11650.644,E2 11650.644} C_VEL
LIN {X 0,Y 562.635,Z 1030.696,A -85,B 0,C 180,E1 11655.393,E2 11655.393} C_VEL
LIN {X 0,Y 573.491,Z 961.378,A -85,B 0,C 180,E1 11658.371,E2 11658.371} C_VEL
LIN {X 0,Y 574.136,Z 943.548,A -85,B 0,C 180,E1 11659.077,E2 11659.077} C_VEL
LIN {X 0,Y 543.482,Z 887.832,A -85,B 0,C 180,E1 11664.941,E2 11664.941} C_VEL
LIN {X 0,Y 513.935,Z 844.06,A -85,B 0,C 180,E1 11671.382,E2 11671.382} C_VEL
LIN {X 0,Y 514.168,Z 844.06,A -85,B 0,C 180,E1 11680.136,E2 11680.136} C_VEL
LIN {X 0,Y 514.998,Z 844.06,A -85,B 0,C 180,E1 11688.934,E2 11688.934} C_VEL
LIN {X 0,Y 514.685,Z 844.06,A -85,B 0,C 180,E1 11699.128,E2 11699.128} C_VEL
LIN {X 0,Y 514.415,Z 844.06,A -85,B 0,C 180,E1 11707.598,E2 11707.598} C_VEL
LIN {X 0,Y 514.044,Z 844.06,A -85,B 0,C 180,E1 11716.5,E2 11716.5} C_VEL
LIN {X 0,Y 513.743,Z 844.06,A -85,B 0,C 180,E1 11725.797,E2 11725.797} C_VEL
LIN {X 0,Y 513.984,Z 845.517,A -85,B 0,C 180,E1 11728.636,E2 11728.636} C_VEL
LIN {X 0,Y 550.362,Z 898.897,A -85,B 0,C 180,E1 11736.129,E2 11736.129} C_VEL
LIN {X 0,Y 575.903,Z 947.813,A -85,B 0,C 180,E1 11740.935,E2 11740.935} C_VEL
LIN {X 0,Y 566.058,Z 1018.354,A -85,B 0,C 180,E1 11743.48,E2 11743.48} C_VEL
LIN {X 0,Y 552.22,Z 1090.422,A -85,B 0,C 180,E1 11747.814,E2 11747.814} C_VEL
LIN {X 0,Y 538.19,Z 1153.885,A -85,B 0,C 180,E1 11753.69,E2 11753.69} C_VEL
LIN {X 0,Y 526.601,Z 1206.804,A -85,B 0,C 180,E1 11760.923,E2 11760.923} C_VEL
LIN {X 0,Y 521.219,Z 1233.551,A -85,B 0,C 180,E1 11765.954,E2 11765.954} C_VEL
LIN {X 0,Y 510.827,Z 1249.117,A -85,B 0,C 180,E1 11769.32,E2 11769.32} C_VEL
LIN {X 0,Y 507.701,Z 1272.256,A -85,B 0,C 180,E1 11777.054,E2 11777.054} C_VEL
LIN {X 0,Y 507.004,Z 1283.765,A -85,B 0,C 180,E1 11783.991,E2 11783.991} C_VEL
LIN {X 0,Y 506.692,Z 1286.837,A -85,B 0,C 180,E1 11790.857,E2 11790.857} C_VEL
LIN {X 0,Y 507.434,Z 1280.487,A -85,B 0,C 180,E1 11798.594,E2 11798.594} C_VEL
LIN {X 0,Y 509.199,Z 1261.058,A -85,B 0,C 180,E1 11807.144,E2 11807.144} C_VEL
LIN {X 0,Y 514.129,Z 1229.358,A -85,B 0,C 180,E1 11815.322,E2 11815.322} C_VEL
LIN {X 0,Y 524.266,Z 1183.206,A -85,B 0,C 180,E1 11823.156,E2 11823.156} C_VEL
LIN {X 0,Y 538.489,Z 1123.985,A -85,B 0,C 180,E1 11829.927,E2 11829.927} C_VEL
LIN {X 0,Y 553.418,Z 1056.306,A -85,B 0,C 180,E1 11835.074,E2 11835.074} C_VEL
LIN {X 0,Y 566.028,Z 980.85,A -85,B 0,C 180,E1 11838.703,E2 11838.703} C_VEL
LIN {X 0,Y 569.396,Z 947.213,A -85,B 0,C 180,E1 11839.847,E2 11839.847} C_VEL
LIN {X 0,Y 537.803,Z 889.889,A -85,B 0,C 180,E1 11845.993,E2 11845.993} C_VEL
LIN {X 0,Y 507.819,Z 849.128,A -85,B 0,C 180,E1 11852.578,E2 11852.578} C_VEL
LIN {X 0,Y 505.938,Z 844.06,A -85,B 0,C 180,E1 11853.38,E2 11853.38} C_VEL
LIN {X 0,Y 506.053,Z 844.06,A -85,B 0,C 180,E1 11863.483,E2 11863.483} C_VEL
LIN {X 0,Y 506.337,Z 844.06,A -85,B 0,C 180,E1 11872.28,E2 11872.28} C_VEL
LIN {X 0,Y 506.678,Z 844.06,A -85,B 0,C 180,E1 11879.17,E2 11879.17} C_VEL
LIN {X 0,Y 506.394,Z 844.06,A -85,B 0,C 180,E1 11887.776,E2 11887.776} C_VEL
LIN {X 0,Y 506.05,Z 844.06,A -85,B 0,C 180,E1 11896.575,E2 11896.575} C_VEL
LIN {X 0,Y 505.757,Z 844.06,A -85,B 0,C 180,E1 11906.77,E2 11906.77} C_VEL
LIN {X 0,Y 542.184,Z 897.875,A -85,B 0,C 180,E1 11915.033,E2 11915.033} C_VEL
LIN {X 0,Y 569.425,Z 950.365,A -85,B 0,C 180,E1 11920.582,E2 11920.582} C_VEL
LIN {X 0,Y 558.824,Z 1020.809,A -85,B 0,C 180,E1 11923.381,E2 11923.381} C_VEL
LIN {X 0,Y 544.571,Z 1089.877,A -85,B 0,C 180,E1 11927.85,E2 11927.85} C_VEL
LIN {X 0,Y 529.503,Z 1152.528,A -85,B 0,C 180,E1 11934.046,E2 11934.046} C_VEL
LIN {X 0,Y 517.486,Z 1203.487,A -85,B 0,C 180,E1 11941.558,E2 11941.558} C_VEL
LIN {X 0,Y 510.554,Z 1239.885,A -85,B 0,C 180,E1 11949.464,E2 11949.464} C_VEL
LIN {X 0,Y 507.684,Z 1264.284,A -85,B 0,C 180,E1 11957.93,E2 11957.93} C_VEL
LIN {X 0,Y 507.218,Z 1275.378,A -85,B 0,C 180,E1 11965.713,E2 11965.713} C_VEL
LIN {X 0,Y 507.224,Z 1276.355,A -85,B 0,C 180,E1 11972.571,E2 11972.571} C_VEL
LIN {X 0,Y 507.349,Z 1267.508,A -85,B 0,C 180,E1 11980.332,E2 11980.332} C_VEL
LIN {X 0,Y 509.441,Z 1247.665,A -85,B 0,C 180,E1 11988.214,E2 11988.214} C_VEL
LIN {X 0,Y 515.935,Z 1212.001,A -85,B 0,C 180,E1 11996.762,E2 11996.762} C_VEL
LIN {X 0,Y 527.106,Z 1162.711,A -85,B 0,C 180,E1 12004.579,E2 12004.579} C_VEL
LIN {X 0,Y 541.595,Z 1102.406,A -85,B 0,C 180,E1 12011.01,E2 12011.01} C_VEL
LIN {X 0,Y 556.453,Z 1033.344,A -85,B 0,C 180,E1 12015.854,E2 12015.854} C_VEL
LIN {X 0,Y 567.906,Z 963.479,A -85,B 0,C 180,E1 12018.916,E2 12018.916} C_VEL
LIN {X 0,Y 568.331,Z 946.523,A -85,B 0,C 180,E1 12019.628,E2 12019.628} C_VEL
LIN {X 0,Y 537.566,Z 890.12,A -85,B 0,C 180,E1 12025.791,E2 12025.791} C_VEL
LIN {X 0,Y 507.561,Z 848.896,A -85,B 0,C 180,E1 12032.415,E2 12032.415} C_VEL
LIN {X 0,Y 505.928,Z 844.06,A -85,B 0,C 180,E1 12032.997,E2 12032.997} C_VEL
LIN {X 0,Y 506.197,Z 844.06,A -85,B 0,C 180,E1 12041.629,E2 12041.629} C_VEL
LIN {X 0,Y 506.734,Z 844.06,A -85,B 0,C 180,E1 12050.495,E2 12050.495} C_VEL
LIN {X 0,Y 506.687,Z 844.06,A -85,B 0,C 180,E1 12059.114,E2 12059.114} C_VEL
LIN {X 0,Y 506.404,Z 844.06,A -85,B 0,C 180,E1 12067.719,E2 12067.719} C_VEL
LIN {X 0,Y 506.05,Z 844.06,A -85,B 0,C 180,E1 12076.517,E2 12076.517} C_VEL
LIN {X 0,Y 505.726,Z 844.06,A -85,B 0,C 180,E1 12086.237,E2 12086.237} C_VEL
LIN {X 0,Y 506.317,Z 846.95,A -85,B 0,C 180,E1 12087.055,E2 12087.055} C_VEL
LIN {X 0,Y 537.687,Z 890.513,A -85,B 0,C 180,E1 12094.015,E2 12094.015} C_VEL
LIN {X 0,Y 570.403,Z 949.772,A -85,B 0,C 180,E1 12100.37,E2 12100.37} C_VEL
LIN {X 0,Y 559.926,Z 1021.575,A -85,B 0,C 180,E1 12103.034,E2 12103.034} C_VEL
LIN {X 0,Y 545.923,Z 1091.146,A -85,B 0,C 180,E1 12107.292,E2 12107.292} C_VEL
LIN {X 0,Y 531.384,Z 1154.166,A -85,B 0,C 180,E1 12113.199,E2 12113.199} C_VEL
LIN {X 0,Y 519.284,Z 1206.748,A -85,B 0,C 180,E1 12120.474,E2 12120.474} C_VEL
LIN {X 0,Y 511.267,Z 1247.032,A -85,B 0,C 180,E1 12128.793,E2 12128.793} C_VEL
LIN {X 0,Y 510.827,Z 1249.117,A -85,B 0,C 180,E1 12129.32,E2 12129.32} C_VEL
LIN {X 0,Y 501.148,Z 1262.028,A -85,B 0,C 180,E1 12132.902,E2 12132.902} C_VEL
LIN {X 0,Y 499.496,Z 1280.619,A -85,B 0,C 180,E1 12141.367,E2 12141.367} C_VEL
LIN {X 0,Y 498.823,Z 1286.836,A -85,B 0,C 180,E1 12149.129,E2 12149.129} C_VEL
LIN {X 0,Y 499.101,Z 1282.882,A -85,B 0,C 180,E1 12156.981,E2 12156.981} C_VEL
LIN {X 0,Y 500.96,Z 1265.692,A -85,B 0,C 180,E1 12165.81,E2 12165.81} C_VEL
LIN {X 0,Y 505.943,Z 1233.578,A -85,B 0,C 180,E1 12174.812,E2 12174.812} C_VEL
LIN {X 0,Y 516.039,Z 1188.254,A -85,B 0,C 180,E1 12182.934,E2 12182.934} C_VEL
LIN {X 0,Y 530.564,Z 1130.542,A -85,B 0,C 180,E1 12189.874,E2 12189.874} C_VEL
LIN {X 0,Y 546.227,Z 1062.84,A -85,B 0,C 180,E1 12195.286,E2 12195.286} C_VEL
LIN {X 0,Y 559.745,Z 987.882,A -85,B 0,C 180,E1 12199.064,E2 12199.064} C_VEL
LIN {X 0,Y 563.874,Z 951.052,A -85,B 0,C 180,E1 12200.366,E2 12200.366} C_VEL
LIN {X 0,Y 533.954,Z 895.729,A -85,B 0,C 180,E1 12206.45,E2 12206.45} C_VEL
LIN {X 0,Y 501.872,Z 850.968,A -85,B 0,C 180,E1 12213.855,E2 12213.855} C_VEL
LIN {X 0,Y 497.823,Z 844.06,A -85,B 0,C 180,E1 12215.259,E2 12215.259} C_VEL
LIN {X 0,Y 498.045,Z 844.06,A -85,B 0,C 180,E1 12225.024,E2 12225.024} C_VEL
LIN {X 0,Y 498.402,Z 844.06,A -85,B 0,C 180,E1 12233.913,E2 12233.913} C_VEL
LIN {X 0,Y 498.455,Z 844.06,A -85,B 0,C 180,E1 12240.9,E2 12240.9} C_VEL
LIN {X 0,Y 498.279,Z 844.06,A -85,B 0,C 180,E1 12249.668,E2 12249.668} C_VEL
LIN {X 0,Y 497.986,Z 844.06,A -85,B 0,C 180,E1 12258.685,E2 12258.685} C_VEL
LIN {X 0,Y 497.957,Z 845.97,A -85,B 0,C 180,E1 12265.157,E2 12265.157} C_VEL
LIN {X 0,Y 528.354,Z 888.188,A -85,B 0,C 180,E1 12272.542,E2 12272.542} C_VEL
LIN {X 0,Y 559.403,Z 942.593,A -85,B 0,C 180,E1 12279.006,E2 12279.006} C_VEL
LIN {X 0,Y 563.444,Z 956.179,A -85,B 0,C 180,E1 12280.128,E2 12280.128} C_VEL
LIN {X 0,Y 551.597,Z 1029.457,A -85,B 0,C 180,E1 12283.233,E2 12283.233} C_VEL
LIN {X 0,Y 536.726,Z 1096.99,A -85,B 0,C 180,E1 12287.852,E2 12287.852} C_VEL
LIN {X 0,Y 521.107,Z 1159.004,A -85,B 0,C 180,E1 12294.318,E2 12294.318} C_VEL
LIN {X 0,Y 509.046,Z 1208.128,A -85,B 0,C 180,E1 12301.966,E2 12301.966} C_VEL
LIN {X 0,Y 502.247,Z 1243.364,A -85,B 0,C 180,E1 12310.142,E2 12310.142} C_VEL
LIN {X 0,Y 499.715,Z 1266.099,A -85,B 0,C 180,E1 12318.623,E2 12318.623} C_VEL
LIN {X 0,Y 499.21,Z 1275.377,A -85,B 0,C 180,E1 12325.644,E2 12325.644} C_VEL
LIN {X 0,Y 499.217,Z 1276.355,A -85,B 0,C 180,E1 12332.612,E2 12332.612} C_VEL
LIN {X 0,Y 499.391,Z 1267.506,A -85,B 0,C 180,E1 12340.498,E2 12340.498} C_VEL
LIN {X 0,Y 501.947,Z 1246.133,A -85,B 0,C 180,E1 12348.953,E2 12348.953} C_VEL
LIN {X 0,Y 509.312,Z 1208.786,A -85,B 0,C 180,E1 12357.795,E2 12357.795} C_VEL
LIN {X 0,Y 521.106,Z 1159.649,A -85,B 0,C 180,E1 12365.497,E2 12365.497} C_VEL
LIN {X 0,Y 536.078,Z 1099.434,A -85,B 0,C 180,E1 12371.855,E2 12371.855} C_VEL
LIN {X 0,Y 551.474,Z 1030.053,A -85,B 0,C 180,E1 12376.644,E2 12376.644} C_VEL
LIN {X 0,Y 562.931,Z 961.338,A -85,B 0,C 180,E1 12379.606,E2 12379.606} C_VEL
LIN {X 0,Y 562.459,Z 949.311,A -85,B 0,C 180,E1 12380.214,E2 12380.214} C_VEL
LIN {X 0,Y 532.575,Z 894.359,A -85,B 0,C 180,E1 12386.471,E2 12386.471} C_VEL
LIN {X 0,Y 501.723,Z 850.861,A -85,B 0,C 180,E1 12393.663,E2 12393.663} C_VEL
LIN {X 0,Y 497.953,Z 844.06,A -85,B 0,C 180,E1 12395.204,E2 12395.204} C_VEL
LIN {X 0,Y 498.639,Z 844.06,A -85,B 0,C 180,E1 12404.984,E2 12404.984} C_VEL
LIN {X 0,Y 498.473,Z 844.06,A -85,B 0,C 180,E1 12413.857,E2 12413.857} C_VEL
LIN {X 0,Y 498.449,Z 844.06,A -85,B 0,C 180,E1 12420.844,E2 12420.844} C_VEL
LIN {X 0,Y 498.337,Z 844.06,A -85,B 0,C 180,E1 12429.61,E2 12429.61} C_VEL
LIN {X 0,Y 498.031,Z 844.06,A -85,B 0,C 180,E1 12438.623,E2 12438.623} C_VEL
LIN {X 0,Y 497.986,Z 846.079,A -85,B 0,C 180,E1 12445.093,E2 12445.093} C_VEL
LIN {X 0,Y 527.863,Z 887.412,A -85,B 0,C 180,E1 12452.33,E2 12452.33} C_VEL
LIN {X 0,Y 560.114,Z 942.902,A -85,B 0,C 180,E1 12458.857,E2 12458.857} C_VEL
LIN {X 0,Y 564.424,Z 956.463,A -85,B 0,C 180,E1 12459.946,E2 12459.946} C_VEL
LIN {X 0,Y 553.552,Z 1026.407,A -85,B 0,C 180,E1 12462.655,E2 12462.655} C_VEL
LIN {X 0,Y 538.829,Z 1095.589,A -85,B 0,C 180,E1 12467.04,E2 12467.04} C_VEL
LIN {X 0,Y 523.799,Z 1157.668,A -85,B 0,C 180,E1 12473.06,E2 12473.06} C_VEL
LIN {X 0,Y 511.104,Z 1210.665,A -85,B 0,C 180,E1 12480.687,E2 12480.687} C_VEL
LIN {X 0,Y 502.878,Z 1250.238,A -85,B 0,C 180,E1 12489.279,E2 12489.279} C_VEL
LIN {X 0,Y 501.148,Z 1262.028,A -85,B 0,C 180,E1 12492.902,E2 12492.902} C_VEL
LIN {X 0,Y 491.858,Z 1272.385,A -85,B 0,C 180,E1 12496.691,E2 12496.691} C_VEL
LIN {X 0,Y 491.044,Z 1283.759,A -85,B 0,C 180,E1 12503.794,E2 12503.794} C_VEL
LIN {X 0,Y 490.704,Z 1286.836,A -85,B 0,C 180,E1 12510.885,E2 12510.885} C_VEL
LIN {X 0,Y 491.463,Z 1280.759,A -85,B 0,C 180,E1 12518.67,E2 12518.67} C_VEL
LIN {X 0,Y 493.324,Z 1261.719,A -85,B 0,C 180,E1 12527.485,E2 12527.485} C_VEL
LIN {X 0,Y 499.044,Z 1229.259,A -85,B 0,C 180,E1 12536.144,E2 12536.144} C_VEL
LIN {X 0,Y 510.291,Z 1182.944,A -85,B 0,C 180,E1 12544.2,E2 12544.2} C_VEL
LIN {X 0,Y 525.765,Z 1123.906,A -85,B 0,C 180,E1 12551.085,E2 12551.085} C_VEL
LIN {X 0,Y 541.838,Z 1056.508,A -85,B 0,C 180,E1 12556.284,E2 12556.284} C_VEL
LIN {X 0,Y 555.42,Z 981.271,A -85,B 0,C 180,E1 12559.933,E2 12559.933} C_VEL
LIN {X 0,Y 558.077,Z 954.386,A -85,B 0,C 180,E1 12560.934,E2 12560.934} C_VEL
LIN {X 0,Y 530.124,Z 901.463,A -85,B 0,C 180,E1 12566.912,E2 12566.912} C_VEL
LIN {X 0,Y 499.156,Z 857.979,A -85,B 0,C 180,E1 12574.268,E2 12574.268} C_VEL
LIN {X 0,Y 489.771,Z 844.06,A -85,B 0,C 180,E1 12577.252,E2 12577.252} C_VEL
LIN {X 0,Y 490.199,Z 844.06,A -85,B 0,C 180,E1 12587.038,E2 12587.038} C_VEL
LIN {X 0,Y 491.157,Z 844.06,A -85,B 0,C 180,E1 12597.373,E2 12597.373} C_VEL
LIN {X 0,Y 490.67,Z 844.06,A -85,B 0,C 180,E1 12606.241,E2 12606.241} C_VEL
LIN {X 0,Y 490.147,Z 844.06,A -85,B 0,C 180,E1 12615.283,E2 12615.283} C_VEL
LIN {X 0,Y 489.956,Z 845.901,A -85,B 0,C 180,E1 12623.076,E2 12623.076} C_VEL
LIN {X 0,Y 519.432,Z 885.912,A -85,B 0,C 180,E1 12630.89,E2 12630.89} C_VEL
LIN {X 0,Y 549.12,Z 936.735,A -85,B 0,C 180,E1 12637.414,E2 12637.414} C_VEL
LIN {X 0,Y 557.854,Z 959.402,A -85,B 0,C 180,E1 12639.589,E2 12639.589} C_VEL
LIN {X 0,Y 545.234,Z 1033.32,A -85,B 0,C 180,E1 12642.809,E2 12642.809} C_VEL
LIN {X 0,Y 529.746,Z 1100.566,A -85,B 0,C 180,E1 12647.551,E2 12647.551} C_VEL
LIN {X 0,Y 513.853,Z 1160.921,A -85,B 0,C 180,E1 12654.009,E2 12654.009} C_VEL
LIN {X 0,Y 501.325,Z 1209.723,A -85,B 0,C 180,E1 12661.805,E2 12661.805} C_VEL
LIN {X 0,Y 494.243,Z 1244.897,A -85,B 0,C 180,E1 12670.274,E2 12670.274} C_VEL
LIN {X 0,Y 491.713,Z 1266.094,A -85,B 0,C 180,E1 12678.436,E2 12678.436} C_VEL
LIN {X 0,Y 491.201,Z 1275.377,A -85,B 0,C 180,E1 12685.573,E2 12685.573} C_VEL
LIN {X 0,Y 491.23,Z 1276.356,A -85,B 0,C 180,E1 12692.654,E2 12692.654} C_VEL
LIN {X 0,Y 491.423,Z 1267.504,A -85,B 0,C 180,E1 12700.671,E2 12700.671} C_VEL
LIN {X 0,Y 494.191,Z 1246.134,A -85,B 0,C 180,E1 12709.262,E2 12709.262} C_VEL
LIN {X 0,Y 501.891,Z 1209.07,A -85,B 0,C 180,E1 12718.204,E2 12718.204} C_VEL
LIN {X 0,Y 514.358,Z 1159.792,A -85,B 0,C 180,E1 12726.028,E2 12726.028} C_VEL
LIN {X 0,Y 529.922,Z 1099.687,A -85,B 0,C 180,E1 12732.437,E2 12732.437} C_VEL
LIN {X 0,Y 545.657,Z 1031.37,A -85,B 0,C 180,E1 12737.201,E2 12737.201} C_VEL
LIN {X 0,Y 557.59,Z 962.61,A -85,B 0,C 180,E1 12740.201,E2 12740.201} C_VEL
LIN {X 0,Y 556.393,Z 951.825,A -85,B 0,C 180,E1 12740.856,E2 12740.856} C_VEL
LIN {X 0,Y 527.062,Z 897.219,A -85,B 0,C 180,E1 12747.307,E2 12747.307} C_VEL
LIN {X 0,Y 498.325,Z 857.198,A -85,B 0,C 180,E1 12754.26,E2 12754.26} C_VEL
LIN {X 0,Y 490.012,Z 844.06,A -85,B 0,C 180,E1 12757.202,E2 12757.202} C_VEL
LIN {X 0,Y 490.897,Z 844.06,A -85,B 0,C 180,E1 12766.689,E2 12766.689} C_VEL
LIN {X 0,Y 491.183,Z 844.06,A -85,B 0,C 180,E1 12777.316,E2 12777.316} C_VEL
LIN {X 0,Y 490.666,Z 844.06,A -85,B 0,C 180,E1 12786.183,E2 12786.183} C_VEL
LIN {X 0,Y 490.16,Z 844.06,A -85,B 0,C 180,E1 12795.223,E2 12795.223} C_VEL
LIN {X 0,Y 490.024,Z 845.924,A -85,B 0,C 180,E1 12803.029,E2 12803.029} C_VEL
LIN {X 0,Y 519.537,Z 886.088,A -85,B 0,C 180,E1 12810.82,E2 12810.82} C_VEL
LIN {X 0,Y 550.532,Z 938.521,A -85,B 0,C 180,E1 12817.431,E2 12817.431} C_VEL
LIN {X 0,Y 558.89,Z 959.18,A -85,B 0,C 180,E1 12819.395,E2 12819.395} C_VEL
LIN {X 0,Y 547.438,Z 1029.638,A -85,B 0,C 180,E1 12822.2,E2 12822.2} C_VEL
LIN {X 0,Y 531.827,Z 1099.713,A -85,B 0,C 180,E1 12826.773,E2 12826.773} C_VEL
LIN {X 0,Y 516.11,Z 1161.416,A -85,B 0,C 180,E1 12832.96,E2 12832.96} C_VEL
LIN {X 0,Y 503.272,Z 1212.52,A -85,B 0,C 180,E1 12840.571,E2 12840.571} C_VEL
LIN {X 0,Y 494.841,Z 1251.677,A -85,B 0,C 180,E1 12849.363,E2 12849.363} C_VEL
LIN {X 0,Y 491.858,Z 1272.385,A -85,B 0,C 180,E1 12856.691,E2 12856.691} C_VEL
LIN {X 0,Y 483.501,Z 1279.996,A -85,B 0,C 180,E1 12860.652,E2 12860.652} C_VEL
LIN {X 0,Y 482.856,Z 1286.836,A -85,B 0,C 180,E1 12869.1,E2 12869.1} C_VEL
LIN {X 0,Y 483.172,Z 1282.882,A -85,B 0,C 180,E1 12877.212,E2 12877.212} C_VEL
LIN {X 0,Y 485.181,Z 1265.691,A -85,B 0,C 180,E1 12886.339,E2 12886.339} C_VEL
LIN {X 0,Y 490.331,Z 1235.386,A -85,B 0,C 180,E1 12895.168,E2 12895.168} C_VEL
LIN {X 0,Y 501.34,Z 1190.347,A -85,B 0,C 180,E1 12903.625,E2 12903.625} C_VEL
LIN {X 0,Y 516.965,Z 1133.487,A -85,B 0,C 180,E1 12910.735,E2 12910.735} C_VEL
LIN {X 0,Y 533.296,Z 1068.576,A -85,B 0,C 180,E1 12916.153,E2 12916.153} C_VEL
LIN {X 0,Y 548.172,Z 994.46,A -85,B 0,C 180,E1 12920.072,E2 12920.072} C_VEL
LIN {X 0,Y 552.434,Z 957.689,A -85,B 0,C 180,E1 12921.498,E2 12921.498} C_VEL
LIN {X 0,Y 525.688,Z 906.171,A -85,B 0,C 180,E1 12927.52,E2 12927.52} C_VEL
LIN {X 0,Y 496.25,Z 864.613,A -85,B 0,C 180,E1 12934.75,E2 12934.75} C_VEL
LIN {X 0,Y 481.873,Z 844.06,A -85,B 0,C 180,E1 12939.77,E2 12939.77} C_VEL
LIN {X 0,Y 482.379,Z 844.06,A -85,B 0,C 180,E1 12950.069,E2 12950.069} C_VEL
LIN {X 0,Y 482.7,Z 844.06,A -85,B 0,C 180,E1 12959.129,E2 12959.129} C_VEL
LIN {X 0,Y 482.335,Z 844.06,A -85,B 0,C 180,E1 12968.166,E2 12968.166} C_VEL
LIN {X 0,Y 481.975,Z 844.06,A -85,B 0,C 180,E1 12977.429,E2 12977.429} C_VEL
LIN {X 0,Y 482.22,Z 846.174,A -85,B 0,C 180,E1 12980.819,E2 12980.819} C_VEL
LIN {X 0,Y 508.281,Z 880.861,A -85,B 0,C 180,E1 12988.565,E2 12988.565} C_VEL
LIN {X 0,Y 537.3,Z 927.706,A -85,B 0,C 180,E1 12995.328,E2 12995.328} C_VEL
LIN {X 0,Y 552.307,Z 962.718,A -85,B 0,C 180,E1 12999.042,E2 12999.042} C_VEL
LIN {X 0,Y 539.002,Z 1036.855,A -85,B 0,C 180,E1 13002.361,E2 13002.361} C_VEL
LIN {X 0,Y 522.456,Z 1105.605,A -85,B 0,C 180,E1 13007.373,E2 13007.373} C_VEL
LIN {X 0,Y 505.889,Z 1165.578,A -85,B 0,C 180,E1 13014.06,E2 13014.06} C_VEL
LIN {X 0,Y 492.957,Z 1214.345,A -85,B 0,C 180,E1 13022.27,E2 13022.27} C_VEL
LIN {X 0,Y 486.005,Z 1249.145,A -85,B 0,C 180,E1 13031.294,E2 13031.294} C_VEL
LIN {X 0,Y 483.567,Z 1269.225,A -85,B 0,C 180,E1 13040.068,E2 13040.068} C_VEL
LIN {X 0,Y 482.89,Z 1276.408,A -85,B 0,C 180,E1 13047.3,E2 13047.3} C_VEL
LIN {X 0,Y 483.154,Z 1275.324,A -85,B 0,C 180,E1 13054.501,E2 13054.501} C_VEL
LIN {X 0,Y 484.371,Z 1262.161,A -85,B 0,C 180,E1 13063.581,E2 13063.581} C_VEL
LIN {X 0,Y 488.326,Z 1234.827,A -85,B 0,C 180,E1 13072.842,E2 13072.842} C_VEL
LIN {X 0,Y 497.673,Z 1195.628,A -85,B 0,C 180,E1 13081.192,E2 13081.192} C_VEL
LIN {X 0,Y 512.479,Z 1141.909,A -85,B 0,C 180,E1 13088.811,E2 13088.811} C_VEL
LIN {X 0,Y 529.281,Z 1078.613,A -85,B 0,C 180,E1 13094.766,E2 13094.766} C_VEL
LIN {X 0,Y 544.842,Z 1006.39,A -85,B 0,C 180,E1 13099.15,E2 13099.15} C_VEL
LIN {X 0,Y 551.779,Z 957.661,A -85,B 0,C 180,E1 13101.173,E2 13101.173} C_VEL
LIN {X 0,Y 523.519,Z 903.323,A -85,B 0,C 180,E1 13107.735,E2 13107.735} C_VEL
LIN {X 0,Y 495.203,Z 863.39,A -85,B 0,C 180,E1 13114.815,E2 13114.815} C_VEL
LIN {X 0,Y 482.093,Z 844.06,A -85,B 0,C 180,E1 13119.236,E2 13119.236} C_VEL
LIN {X 0,Y 482.905,Z 844.06,A -85,B 0,C 180,E1 13128.188,E2 13128.188} C_VEL
LIN {X 0,Y 482.709,Z 844.06,A -85,B 0,C 180,E1 13139.07,E2 13139.07} C_VEL
LIN {X 0,Y 482.365,Z 844.06,A -85,B 0,C 180,E1 13148.107,E2 13148.107} C_VEL
LIN {X 0,Y 481.975,Z 844.06,A -85,B 0,C 180,E1 13157.368,E2 13157.368} C_VEL
LIN {X 0,Y 482.207,Z 846.148,A -85,B 0,C 180,E1 13160.757,E2 13160.757} C_VEL
LIN {X 0,Y 508.801,Z 881.687,A -85,B 0,C 180,E1 13168.611,E2 13168.611} C_VEL
LIN {X 0,Y 538.562,Z 929.335,A -85,B 0,C 180,E1 13175.359,E2 13175.359} C_VEL
LIN {X 0,Y 553.221,Z 963.202,A -85,B 0,C 180,E1 13178.871,E2 13178.871} C_VEL
LIN {X 0,Y 541.216,Z 1033.27,A -85,B 0,C 180,E1 13181.763,E2 13181.763} C_VEL
LIN {X 0,Y 525.106,Z 1102.253,A -85,B 0,C 180,E1 13186.377,E2 13186.377} C_VEL
LIN {X 0,Y 508.939,Z 1163.088,A -85,B 0,C 180,E1 13192.617,E2 13192.617} C_VEL
LIN {X 0,Y 495.614,Z 1213.808,A -85,B 0,C 180,E1 13200.358,E2 13200.358} C_VEL
LIN {X 0,Y 487.127,Z 1251.654,A -85,B 0,C 180,E1 13209.021,E2 13209.021} C_VEL
LIN {X 0,Y 483.687,Z 1274.184,A -85,B 0,C 180,E1 13217.322,E2 13217.322} C_VEL
LIN {X 0,Y 483.501,Z 1279.996,A -85,B 0,C 180,E1 13220.652,E2 13220.652} C_VEL
LIN {X 0,Y 475.073,Z 1284.759,A -85,B 0,C 180,E1 13224.743,E2 13224.743} C_VEL
LIN {X 0,Y 475.143,Z 1286.382,A -85,B 0,C 180,E1 13232.744,E2 13232.744} C_VEL
LIN {X 0,Y 475.566,Z 1277.577,A -85,B 0,C 180,E1 13241.031,E2 13241.031} C_VEL
LIN {X 0,Y 478.321,Z 1256.471,A -85,B 0,C 180,E1 13249.845,E2 13249.845} C_VEL
LIN {X 0,Y 486.036,Z 1221.35,A -85,B 0,C 180,E1 13258.668,E2 13258.668} C_VEL
LIN {X 0,Y 499.654,Z 1171.816,A -85,B 0,C 180,E1 13266.83,E2 13266.83} C_VEL
LIN {X 0,Y 516.64,Z 1111.47,A -85,B 0,C 180,E1 13273.457,E2 13273.457} C_VEL
LIN {X 0,Y 533.386,Z 1044.329,A -85,B 0,C 180,E1 13278.29,E2 13278.29} C_VEL
LIN {X 0,Y 547.065,Z 970.395,A -85,B 0,C 180,E1 13281.587,E2 13281.587} C_VEL
LIN {X 0,Y 546.478,Z 960.454,A -85,B 0,C 180,E1 13282.149,E2 13282.149} C_VEL
LIN {X 0,Y 520.696,Z 909.796,A -85,B 0,C 180,E1 13288.28,E2 13288.28} C_VEL
LIN {X 0,Y 492.772,Z 870.414,A -85,B 0,C 180,E1 13295.42,E2 13295.42} C_VEL
LIN {X 0,Y 476.53,Z 849.97,A -85,B 0,C 180,E1 13301.005,E2 13301.005} C_VEL
LIN {X 0,Y 473.937,Z 844.06,A -85,B 0,C 180,E1 13302.328,E2 13302.328} C_VEL
LIN {X 0,Y 474.309,Z 844.06,A -85,B 0,C 180,E1 13311.755,E2 13311.755} C_VEL
LIN {X 0,Y 474.716,Z 844.06,A -85,B 0,C 180,E1 13319.114,E2 13319.114} C_VEL
LIN {X 0,Y 474.312,Z 844.06,A -85,B 0,C 180,E1 13328.305,E2 13328.305} C_VEL
LIN {X 0,Y 474.114,Z 845.77,A -85,B 0,C 180,E1 13338.039,E2 13338.039} C_VEL
LIN {X 0,Y 496.861,Z 875.816,A -85,B 0,C 180,E1 13345.874,E2 13345.874} C_VEL
LIN {X 0,Y 526.13,Z 920.252,A -85,B 0,C 180,E1 13353.251,E2 13353.251} C_VEL
LIN {X 0,Y 547.02,Z 964.335,A -85,B 0,C 180,E1 13358.437,E2 13358.437} C_VEL
LIN {X 0,Y 533.151,Z 1038.661,A -85,B 0,C 180,E1 13361.811,E2 13361.811} C_VEL
LIN {X 0,Y 516.154,Z 1106.52,A -85,B 0,C 180,E1 13366.825,E2 13366.825} C_VEL
LIN {X 0,Y 498.823,Z 1166.675,A -85,B 0,C 180,E1 13373.641,E2 13373.641} C_VEL
LIN {X 0,Y 485.509,Z 1214.433,A -85,B 0,C 180,E1 13381.807,E2 13381.807} C_VEL
LIN {X 0,Y 478.268,Z 1248.015,A -85,B 0,C 180,E1 13390.553,E2 13390.553} C_VEL
LIN {X 0,Y 475.587,Z 1269.22,A -85,B 0,C 180,E1 13399.899,E2 13399.899} C_VEL
LIN {X 0,Y 474.893,Z 1276.407,A -85,B 0,C 180,E1 13407.254,E2 13407.254} C_VEL
LIN {X 0,Y 475.166,Z 1275.324,A -85,B 0,C 180,E1 13414.577,E2 13414.577} C_VEL
LIN {X 0,Y 476.43,Z 1262.163,A -85,B 0,C 180,E1 13423.812,E2 13423.812} C_VEL
LIN {X 0,Y 480.643,Z 1234.921,A -85,B 0,C 180,E1 13433.229,E2 13433.229} C_VEL
LIN {X 0,Y 490.656,Z 1195.189,A -85,B 0,C 180,E1 13441.795,E2 13441.795} C_VEL
LIN {X 0,Y 506.268,Z 1140.931,A -85,B 0,C 180,E1 13449.535,E2 13449.535} C_VEL
LIN {X 0,Y 523.741,Z 1077.718,A -85,B 0,C 180,E1 13455.476,E2 13455.476} C_VEL
LIN {X 0,Y 539.578,Z 1006.404,A -85,B 0,C 180,E1 13459.807,E2 13459.807} C_VEL
LIN {X 0,Y 546.33,Z 961.359,A -85,B 0,C 180,E1 13461.712,E2 13461.712} C_VEL
LIN {X 0,Y 519.233,Z 908.485,A -85,B 0,C 180,E1 13468.301,E2 13468.301} C_VEL
LIN {X 0,Y 490.131,Z 866.01,A -85,B 0,C 180,E1 13476.02,E2 13476.02} C_VEL
LIN {X 0,Y 474.201,Z 844.06,A -85,B 0,C 180,E1 13482.276,E2 13482.276} C_VEL
LIN {X 0,Y 474.755,Z 844.06,A -85,B 0,C 180,E1 13489.848,E2 13489.848} C_VEL
LIN {X 0,Y 474.726,Z 844.06,A -85,B 0,C 180,E1 13499.055,E2 13499.055} C_VEL
LIN {X 0,Y 474.344,Z 844.06,A -85,B 0,C 180,E1 13508.245,E2 13508.245} C_VEL
LIN {X 0,Y 474.057,Z 845.583,A -85,B 0,C 180,E1 13517.968,E2 13517.968} C_VEL
LIN {X 0,Y 497.027,Z 876.122,A -85,B 0,C 180,E1 13525.847,E2 13525.847} C_VEL
LIN {X 0,Y 525.144,Z 918.216,A -85,B 0,C 180,E1 13532.825,E2 13532.825} C_VEL
LIN {X 0,Y 547.917,Z 965.013,A -85,B 0,C 180,E1 13538.27,E2 13538.27} C_VEL
LIN {X 0,Y 535.41,Z 1034.926,A -85,B 0,C 180,E1 13541.204,E2 13541.204} C_VEL
LIN {X 0,Y 518.755,Z 1103.477,A -85,B 0,C 180,E1 13545.856,E2 13545.856} C_VEL
LIN {X 0,Y 501.789,Z 1164.759,A -85,B 0,C 180,E1 13552.265,E2 13552.265} C_VEL
LIN {X 0,Y 487.583,Z 1216.26,A -85,B 0,C 180,E1 13560.359,E2 13560.359} C_VEL
LIN {X 0,Y 478.874,Z 1253.874,A -85,B 0,C 180,E1 13569.368,E2 13569.368} C_VEL
LIN {X 0,Y 475.539,Z 1276.01,A -85,B 0,C 180,E1 13578.036,E2 13578.036} C_VEL
LIN {X 0,Y 475.073,Z 1284.759,A -85,B 0,C 180,E1 13584.743,E2 13584.743} C_VEL
LIN {X 0,Y 466.868,Z 1286.809,A -85,B 0,C 180,E1 13588.958,E2 13588.958} C_VEL
LIN {X 0,Y 467.08,Z 1283.752,A -85,B 0,C 180,E1 13596.525,E2 13596.525} C_VEL
LIN {X 0,Y 468.844,Z 1269.082,A -85,B 0,C 180,E1 13605.477,E2 13605.477} C_VEL
LIN {X 0,Y 474.291,Z 1240.076,A -85,B 0,C 180,E1 13614.825,E2 13614.825} C_VEL
LIN {X 0,Y 485.794,Z 1195.989,A -85,B 0,C 180,E1 13623.78,E2 13623.78} C_VEL
LIN {X 0,Y 502.467,Z 1139.916,A -85,B 0,C 180,E1 13631.269,E2 13631.269} C_VEL
LIN {X 0,Y 520.541,Z 1074.138,A -85,B 0,C 180,E1 13637.063,E2 13637.063} C_VEL
LIN {X 0,Y 536.909,Z 999.718,A -85,B 0,C 180,E1 13641.17,E2 13641.17} C_VEL
LIN {X 0,Y 541.492,Z 965.156,A -85,B 0,C 180,E1 13642.594,E2 13642.594} C_VEL
LIN {X 0,Y 516.613,Z 915.271,A -85,B 0,C 180,E1 13648.802,E2 13648.802} C_VEL
LIN {X 0,Y 487.869,Z 873.435,A -85,B 0,C 180,E1 13656.598,E2 13656.598} C_VEL
LIN {X 0,Y 469.523,Z 850.744,A -85,B 0,C 180,E1 13663.619,E2 13663.619} C_VEL
LIN {X 0,Y 466.054,Z 844.06,A -85,B 0,C 180,E1 13665.901,E2 13665.901} C_VEL
LIN {X 0,Y 466.719,Z 844.06,A -85,B 0,C 180,E1 13675.369,E2 13675.369} C_VEL
LIN {X 0,Y 466.859,Z 844.06,A -85,B 0,C 180,E1 13684.69,E2 13684.69} C_VEL
LIN {X 0,Y 466.313,Z 845.967,A -85,B 0,C 180,E1 13694.815,E2 13694.815} C_VEL
LIN {X 0,Y 483.633,Z 868.294,A -85,B 0,C 180,E1 13702.128,E2 13702.128} C_VEL
LIN {X 0,Y 510.575,Z 906.414,A -85,B 0,C 180,E1 13709.878,E2 13709.878} C_VEL
LIN {X 0,Y 536.883,Z 956.208,A -85,B 0,C 180,E1 13716.618,E2 13716.618} C_VEL
LIN {X 0,Y 541.165,Z 969.335,A -85,B 0,C 180,E1 13717.937,E2 13717.937} C_VEL
LIN {X 0,Y 526.874,Z 1042.212,A -85,B 0,C 180,E1 13721.361,E2 13721.361} C_VEL
LIN {X 0,Y 509.176,Z 1109.794,A -85,B 0,C 180,E1 13726.494,E2 13726.494} C_VEL
LIN {X 0,Y 491.387,Z 1169.042,A -85,B 0,C 180,E1 13733.395,E2 13733.395} C_VEL
LIN {X 0,Y 477.617,Z 1216.679,A -85,B 0,C 180,E1 13741.816,E2 13741.816} C_VEL
LIN {X 0,Y 470.131,Z 1250.761,A -85,B 0,C 180,E1 13751.181,E2 13751.181} C_VEL
LIN {X 0,Y 467.439,Z 1270.53,A -85,B 0,C 180,E1 13760.664,E2 13760.664} C_VEL
LIN {X 0,Y 466.976,Z 1276.844,A -85,B 0,C 180,E1 13769.07,E2 13769.07} C_VEL
LIN {X 0,Y 467.42,Z 1273.709,A -85,B 0,C 180,E1 13776.52,E2 13776.52} C_VEL
LIN {X 0,Y 468.598,Z 1259.09,A -85,B 0,C 180,E1 13785.486,E2 13785.486} C_VEL
LIN {X 0,Y 473.852,Z 1231.205,A -85,B 0,C 180,E1 13794.664,E2 13794.664} C_VEL
LIN {X 0,Y 484.972,Z 1190.497,A -85,B 0,C 180,E1 13803.178,E2 13803.178} C_VEL
LIN {X 0,Y 501.652,Z 1135.146,A -85,B 0,C 180,E1 13810.824,E2 13810.824} C_VEL
LIN {X 0,Y 519.967,Z 1070.406,A -85,B 0,C 180,E1 13816.678,E2 13816.678} C_VEL
LIN {X 0,Y 536.041,Z 997.876,A -85,B 0,C 180,E1 13820.867,E2 13820.867} C_VEL
LIN {X 0,Y 541.331,Z 966.227,A -85,B 0,C 180,E1 13822.125,E2 13822.125} C_VEL
LIN {X 0,Y 515.535,Z 914.492,A -85,B 0,C 180,E1 13828.727,E2 13828.727} C_VEL
LIN {X 0,Y 487.801,Z 873.199,A -85,B 0,C 180,E1 13836.385,E2 13836.385} C_VEL
LIN {X 0,Y 469.424,Z 850.416,A -85,B 0,C 180,E1 13843.398,E2 13843.398} C_VEL
LIN {X 0,Y 466.583,Z 844.06,A -85,B 0,C 180,E1 13845.374,E2 13845.374} C_VEL
LIN {X 0,Y 466.765,Z 844.06,A -85,B 0,C 180,E1 13855.309,E2 13855.309} C_VEL
LIN {X 0,Y 466.84,Z 844.06,A -85,B 0,C 180,E1 13864.63,E2 13864.63} C_VEL
LIN {X 0,Y 466.335,Z 846.002,A -85,B 0,C 180,E1 13874.812,E2 13874.812} C_VEL
LIN {X 0,Y 483.859,Z 868.646,A -85,B 0,C 180,E1 13882.145,E2 13882.145} C_VEL
LIN {X 0,Y 510.617,Z 906.252,A -85,B 0,C 180,E1 13889.751,E2 13889.751} C_VEL
LIN {X 0,Y 537.923,Z 956.91,A -85,B 0,C 180,E1 13896.496,E2 13896.496} C_VEL
LIN {X 0,Y 542.185,Z 970.485,A -85,B 0,C 180,E1 13897.774,E2 13897.774} C_VEL
LIN {X 0,Y 528.654,Z 1040.997,A -85,B 0,C 180,E1 13900.87,E2 13900.87} C_VEL
LIN {X 0,Y 511.035,Z 1109.965,A -85,B 0,C 180,E1 13905.783,E2 13905.783} C_VEL
LIN {X 0,Y 493.59,Z 1169.958,A -85,B 0,C 180,E1 13912.363,E2 13912.363} C_VEL
LIN {X 0,Y 479.204,Z 1220.054,A -85,B 0,C 180,E1 13920.625,E2 13920.625} C_VEL
LIN {X 0,Y 470.809,Z 1255.301,A -85,B 0,C 180,E1 13929.482,E2 13929.482} C_VEL
LIN {X 0,Y 467.6,Z 1276.007,A -85,B 0,C 180,E1 13937.83,E2 13937.83} C_VEL
LIN {X 0,Y 467.145,Z 1285.349,A -85,B 0,C 180,E1 13945.345,E2 13945.345} C_VEL
LIN {X 0,Y 466.868,Z 1286.809,A -85,B 0,C 180,E1 13948.958,E2 13948.958} C_VEL
LIN {X 0,Y 459.1,Z 1286.166,A -85,B 0,C 180,E1 13953.236,E2 13953.236} C_VEL
LIN {X 0,Y 459.674,Z 1275.921,A -85,B 0,C 180,E1 13962.383,E2 13962.383} C_VEL
LIN {X 0,Y 463.592,Z 1253.136,A -85,B 0,C 180,E1 13971.526,E2 13971.526} C_VEL
LIN {X 0,Y 473.38,Z 1215.113,A -85,B 0,C 180,E1 13980.836,E2 13980.836} C_VEL
LIN {X 0,Y 488.645,Z 1164.283,A -85,B 0,C 180,E1 13988.985,E2 13988.985} C_VEL
LIN {X 0,Y 507.097,Z 1102.953,A -85,B 0,C 180,E1 13995.482,E2 13995.482} C_VEL
LIN {X 0,Y 524.957,Z 1033.874,A -85,B 0,C 180,E1 14000.195,E2 14000.195} C_VEL
LIN {X 0,Y 536.149,Z 968.94,A -85,B 0,C 180,E1 14003.148,E2 14003.148} C_VEL
LIN {X 0,Y 512.173,Z 919.986,A -85,B 0,C 180,E1 14009.429,E2 14009.429} C_VEL
LIN {X 0,Y 485.098,Z 880.188,A -85,B 0,C 180,E1 14017.112,E2 14017.112} C_VEL
LIN {X 0,Y 467.618,Z 858.091,A -85,B 0,C 180,E1 14024.024,E2 14024.024} C_VEL
LIN {X 0,Y 461.297,Z 850.344,A -85,B 0,C 180,E1 14027.568,E2 14027.568} C_VEL
LIN {X 0,Y 458.267,Z 844.06,A -85,B 0,C 180,E1 14030.504,E2 14030.504} C_VEL
LIN {X 0,Y 458.718,Z 844.06,A -85,B 0,C 180,E1 14039.083,E2 14039.083} C_VEL
LIN {X 0,Y 458.291,Z 844.06,A -85,B 0,C 180,E1 14048.598,E2 14048.598} C_VEL
LIN {X 0,Y 458.705,Z 846.799,A -85,B 0,C 180,E1 14050.692,E2 14050.692} C_VEL
LIN {X 0,Y 465.648,Z 855.681,A -85,B 0,C 180,E1 14055.078,E2 14055.078} C_VEL
LIN {X 0,Y 481.26,Z 874.99,A -85,B 0,C 180,E1 14061.688,E2 14061.688} C_VEL
LIN {X 0,Y 507.359,Z 913.038,A -85,B 0,C 180,E1 14069.532,E2 14069.532} C_VEL
LIN {X 0,Y 532.448,Z 962.007,A -85,B 0,C 180,E1 14076.273,E2 14076.273} C_VEL
LIN {X 0,Y 535.45,Z 973.951,A -85,B 0,C 180,E1 14077.417,E2 14077.417} C_VEL
LIN {X 0,Y 519.918,Z 1048.556,A -85,B 0,C 180,E1 14081.07,E2 14081.07} C_VEL
LIN {X 0,Y 501.431,Z 1115.714,A -85,B 0,C 180,E1 14086.412,E2 14086.412} C_VEL
LIN {X 0,Y 483.222,Z 1173.822,A -85,B 0,C 180,E1 14093.5,E2 14093.5} C_VEL
LIN {X 0,Y 469.429,Z 1220.005,A -85,B 0,C 180,E1 14102.067,E2 14102.067} C_VEL
LIN {X 0,Y 461.977,Z 1253.504,A -85,B 0,C 180,E1 14111.829,E2 14111.829} C_VEL
LIN {X 0,Y 459.285,Z 1271.771,A -85,B 0,C 180,E1 14121.455,E2 14121.455} C_VEL
LIN {X 0,Y 458.972,Z 1276.844,A -85,B 0,C 180,E1 14129.053,E2 14129.053} C_VEL
LIN {X 0,Y 459.426,Z 1272.501,A -85,B 0,C 180,E1 14137.868,E2 14137.868} C_VEL
LIN {X 0,Y 460.917,Z 1256.595,A -85,B 0,C 180,E1 14146.866,E2 14146.866} C_VEL
LIN {X 0,Y 466.69,Z 1229.662,A -85,B 0,C 180,E1 14155.504,E2 14155.504} C_VEL
LIN {X 0,Y 478.836,Z 1187.684,A -85,B 0,C 180,E1 14164.21,E2 14164.21} C_VEL
LIN {X 0,Y 496.36,Z 1132.103,A -85,B 0,C 180,E1 14171.792,E2 14171.792} C_VEL
LIN {X 0,Y 514.815,Z 1068.797,A -85,B 0,C 180,E1 14177.463,E2 14177.463} C_VEL
LIN {X 0,Y 531.369,Z 996.006,A -85,B 0,C 180,E1 14181.624,E2 14181.624} C_VEL
LIN {X 0,Y 535.704,Z 969.492,A -85,B 0,C 180,E1 14182.716,E2 14182.716} C_VEL
LIN {X 0,Y 510.2,Z 917.49,A -85,B 0,C 180,E1 14189.605,E2 14189.605} C_VEL
LIN {X 0,Y 484.17,Z 879.075,A -85,B 0,C 180,E1 14197.171,E2 14197.171} C_VEL
LIN {X 0,Y 467.462,Z 857.654,A -85,B 0,C 180,E1 14203.832,E2 14203.832} C_VEL
LIN {X 0,Y 461.915,Z 850.469,A -85,B 0,C 180,E1 14206.904,E2 14206.904} C_VEL
LIN {X 0,Y 458.744,Z 844.06,A -85,B 0,C 180,E1 14209.489,E2 14209.489} C_VEL
LIN {X 0,Y 458.728,Z 844.06,A -85,B 0,C 180,E1 14219.022,E2 14219.022} C_VEL
LIN {X 0,Y 458.31,Z 844.06,A -85,B 0,C 180,E1 14228.535,E2 14228.535} C_VEL
LIN {X 0,Y 458.67,Z 846.578,A -85,B 0,C 180,E1 14230.691,E2 14230.691} C_VEL
LIN {X 0,Y 465.776,Z 855.908,A -85,B 0,C 180,E1 14235.132,E2 14235.132} C_VEL
LIN {X 0,Y 481.3,Z 874.991,A -85,B 0,C 180,E1 14241.64,E2 14241.64} C_VEL
LIN {X 0,Y 508.103,Z 913.893,A -85,B 0,C 180,E1 14249.544,E2 14249.544} C_VEL
LIN {X 0,Y 533.941,Z 963.856,A -85,B 0,C 180,E1 14256.281,E2 14256.281} C_VEL
LIN {X 0,Y 536.446,Z 974.98,A -85,B 0,C 180,E1 14257.247,E2 14257.247} C_VEL
LIN {X 0,Y 522.421,Z 1045.029,A -85,B 0,C 180,E1 14260.421,E2 14260.421} C_VEL
LIN {X 0,Y 504.064,Z 1113.67,A -85,B 0,C 180,E1 14265.46,E2 14265.46} C_VEL
LIN {X 0,Y 485.822,Z 1173.483,A -85,B 0,C 180,E1 14272.238,E2 14272.238} C_VEL
LIN {X 0,Y 471.198,Z 1222.334,A -85,B 0,C 180,E1 14280.606,E2 14280.606} C_VEL
LIN {X 0,Y 462.572,Z 1257.565,A -85,B 0,C 180,E1 14289.864,E2 14289.864} C_VEL
LIN {X 0,Y 459.531,Z 1277.503,A -85,B 0,C 180,E1 14298.579,E2 14298.579} C_VEL
LIN {X 0,Y 459.234,Z 1286.381,A -85,B 0,C 180,E1 14307.161,E2 14307.161} C_VEL
LIN {X 0,Y 459.1,Z 1286.166,A -85,B 0,C 180,E1 14313.236,E2 14313.236} C_VEL
LIN {X 0,Y 451.233,Z 1282.923,A -85,B 0,C 180,E1 14317.569,E2 14317.569} C_VEL
LIN {X 0,Y 453.439,Z 1266.369,A -85,B 0,C 180,E1 14327.109,E2 14327.109} C_VEL
LIN {X 0,Y 459.837,Z 1235.904,A -85,B 0,C 180,E1 14336.728,E2 14336.728} C_VEL
LIN {X 0,Y 473.094,Z 1191.966,A -85,B 0,C 180,E1 14345.55,E2 14345.55} C_VEL
LIN {X 0,Y 491.458,Z 1135.156,A -85,B 0,C 180,E1 14353.057,E2 14353.057} C_VEL
LIN {X 0,Y 510.483,Z 1070.518,A -85,B 0,C 180,E1 14358.649,E2 14358.649} C_VEL
LIN {X 0,Y 527.261,Z 997.316,A -85,B 0,C 180,E1 14362.647,E2 14362.647} C_VEL
LIN {X 0,Y 530.88,Z 973.123,A -85,B 0,C 180,E1 14363.667,E2 14363.667} C_VEL
LIN {X 0,Y 508.167,Z 925.323,A -85,B 0,C 180,E1 14369.968,E2 14369.968} C_VEL
LIN {X 0,Y 482.527,Z 886.98,A -85,B 0,C 180,E1 14377.583,E2 14377.583} C_VEL
LIN {X 0,Y 465.383,Z 865.029,A -85,B 0,C 180,E1 14384.613,E2 14384.613} C_VEL
LIN {X 0,Y 455.975,Z 851.725,A -85,B 0,C 180,E1 14390.939,E2 14390.939} C_VEL
LIN {X 0,Y 450.873,Z 846.496,A -85,B 0,C 180,E1 14400.513,E2 14400.513} C_VEL
LIN {X 0,Y 457.356,Z 854.396,A -85,B 0,C 180,E1 14410.422,E2 14410.422} C_VEL
LIN {X 0,Y 468.765,Z 868.463,A -85,B 0,C 180,E1 14417.105,E2 14417.105} C_VEL
LIN {X 0,Y 492.725,Z 901.269,A -85,B 0,C 180,E1 14425.81,E2 14425.81} C_VEL
LIN {X 0,Y 518.477,Z 946.631,A -85,B 0,C 180,E1 14433.213,E2 14433.213} C_VEL
LIN {X 0,Y 530.042,Z 976.941,A -85,B 0,C 180,E1 14436.824,E2 14436.824} C_VEL
LIN {X 0,Y 514.12,Z 1050.426,A -85,B 0,C 180,E1 14440.494,E2 14440.494} C_VEL
LIN {X 0,Y 495.193,Z 1116.669,A -85,B 0,C 180,E1 14445.837,E2 14445.837} C_VEL
LIN {X 0,Y 476.412,Z 1174.196,A -85,B 0,C 180,E1 14452.943,E2 14452.943} C_VEL
LIN {X 0,Y 461.79,Z 1221.107,A -85,B 0,C 180,E1 14461.815,E2 14461.815} C_VEL
LIN {X 0,Y 454.103,Z 1253.592,A -85,B 0,C 180,E1 14471.502,E2 14471.502} C_VEL
LIN {X 0,Y 451.343,Z 1271.858,A -85,B 0,C 180,E1 14481.303,E2 14481.303} C_VEL
LIN {X 0,Y 450.969,Z 1276.912,A -85,B 0,C 180,E1 14489.037,E2 14489.037} C_VEL
LIN {X 0,Y 451.421,Z 1273.331,A -85,B 0,C 180,E1 14497.292,E2 14497.292} C_VEL
LIN {X 0,Y 452.864,Z 1258.135,A -85,B 0,C 180,E1 14506.538,E2 14506.538} C_VEL
LIN {X 0,Y 458.721,Z 1231.693,A -85,B 0,C 180,E1 14515.454,E2 14515.454} C_VEL
LIN {X 0,Y 471.476,Z 1189.252,A -85,B 0,C 180,E1 14524.536,E2 14524.536} C_VEL
LIN {X 0,Y 489.545,Z 1134.285,A -85,B 0,C 180,E1 14532.21,E2 14532.21} C_VEL
LIN {X 0,Y 508.978,Z 1070.152,A -85,B 0,C 180,E1 14538.052,E2 14538.052} C_VEL
LIN {X 0,Y 525.874,Z 998.749,A -85,B 0,C 180,E1 14542.202,E2 14542.202} C_VEL
LIN {X 0,Y 530.031,Z 972.593,A -85,B 0,C 180,E1 14543.345,E2 14543.345} C_VEL
LIN {X 0,Y 506.011,Z 922.743,A -85,B 0,C 180,E1 14550.196,E2 14550.196} C_VEL
LIN {X 0,Y 481.804,Z 885.955,A -85,B 0,C 180,E1 14557.586,E2 14557.586} C_VEL
LIN {X 0,Y 462.248,Z 859.219,A -85,B 0,C 180,E1 14566.154,E2 14566.154} C_VEL
LIN {X 0,Y 455.053,Z 851.272,A -85,B 0,C 180,E1 14571.341,E2 14571.341} C_VEL
LIN {X 0,Y 450.692,Z 845.506,A -85,B 0,C 180,E1 14579.969,E2 14579.969} C_VEL
LIN {X 0,Y 457.374,Z 854.397,A -85,B 0,C 180,E1 14590.48,E2 14590.48} C_VEL
LIN {X 0,Y 468.973,Z 868.891,A -85,B 0,C 180,E1 14597.175,E2 14597.175} C_VEL
LIN {X 0,Y 491.971,Z 900.234,A -85,B 0,C 180,E1 14605.483,E2 14605.483} C_VEL
LIN {X 0,Y 518.014,Z 944.579,A -85,B 0,C 180,E1 14612.773,E2 14612.773} C_VEL
LIN {X 0,Y 531.186,Z 977.07,A -85,B 0,C 180,E1 14616.628,E2 14616.628} C_VEL
LIN {X 0,Y 516.691,Z 1046.793,A -85,B 0,C 180,E1 14619.841,E2 14619.841} C_VEL
LIN {X 0,Y 497.791,Z 1114.792,A -85,B 0,C 180,E1 14624.902,E2 14624.902} C_VEL
LIN {X 0,Y 478.68,Z 1174.917,A -85,B 0,C 180,E1 14631.845,E2 14631.845} C_VEL
LIN {X 0,Y 463.56,Z 1223.332,A -85,B 0,C 180,E1 14640.341,E2 14640.341} C_VEL
LIN {X 0,Y 454.826,Z 1257.475,A -85,B 0,C 180,E1 14649.506,E2 14649.506} C_VEL
LIN {X 0,Y 451.573,Z 1277.414,A -85,B 0,C 180,E1 14658.375,E2 14658.375} C_VEL
LIN {X 0,Y 451.224,Z 1286.313,A -85,B 0,C 180,E1 14667.11,E2 14667.11} C_VEL
LIN {X 0,Y 451.162,Z 1285.27,A -85,B 0,C 180,E1 14674.82,E2 14674.82} C_VEL
LIN {X 0,Y 451.233,Z 1282.923,A -85,B 0,C 180,E1 14677.569,E2 14677.569} C_VEL
LIN {X 0,Y 443.658,Z 1277.124,A -85,B 0,C 180,E1 14681.963,E2 14681.963} C_VEL
LIN {X 0,Y 447.379,Z 1256.179,A -85,B 0,C 180,E1 14691.258,E2 14691.258} C_VEL
LIN {X 0,Y 457.433,Z 1219.775,A -85,B 0,C 180,E1 14700.922,E2 14700.922} C_VEL
LIN {X 0,Y 473.651,Z 1170.178,A -85,B 0,C 180,E1 14709.439,E2 14709.439} C_VEL
LIN {X 0,Y 493.637,Z 1109.12,A -85,B 0,C 180,E1 14716.294,E2 14716.294} C_VEL
LIN {X 0,Y 512.763,Z 1041.725,A -85,B 0,C 180,E1 14721.145,E2 14721.145} C_VEL
LIN {X 0,Y 525.419,Z 976.701,A -85,B 0,C 180,E1 14724.253,E2 14724.253} C_VEL
LIN {X 0,Y 503.657,Z 929.761,A -85,B 0,C 180,E1 14730.666,E2 14730.666} C_VEL
LIN {X 0,Y 479.644,Z 893.346,A -85,B 0,C 180,E1 14738.154,E2 14738.154} C_VEL
LIN {X 0,Y 462.751,Z 871.172,A -85,B 0,C 180,E1 14745.465,E2 14745.465} C_VEL
LIN {X 0,Y 453.919,Z 859.265,A -85,B 0,C 180,E1 14751.866,E2 14751.866} C_VEL
LIN {X 0,Y 449.898,Z 854.437,A -85,B 0,C 180,E1 14760.514,E2 14760.514} C_VEL
LIN {X 0,Y 456.141,Z 862.348,A -85,B 0,C 180,E1 14770.269,E2 14770.269} C_VEL
LIN {X 0,Y 467.399,Z 876.637,A -85,B 0,C 180,E1 14776.978,E2 14776.978} C_VEL
LIN {X 0,Y 490.218,Z 908.482,A -85,B 0,C 180,E1 14785.521,E2 14785.521} C_VEL
LIN {X 0,Y 514.658,Z 953.348,A -85,B 0,C 180,E1 14792.954,E2 14792.954} C_VEL
LIN {X 0,Y 524.558,Z 980.876,A -85,B 0,C 180,E1 14796.258,E2 14796.258} C_VEL
LIN {X 0,Y 507.651,Z 1055.113,A -85,B 0,C 180,E1 14800.083,E2 14800.083} C_VEL
LIN {X 0,Y 487.828,Z 1121.34,A -85,B 0,C 180,E1 14805.616,E2 14805.616} C_VEL
LIN {X 0,Y 468.459,Z 1178.422,A -85,B 0,C 180,E1 14812.965,E2 14812.965} C_VEL
LIN {X 0,Y 453.786,Z 1223.709,A -85,B 0,C 180,E1 14821.923,E2 14821.923} C_VEL
LIN {X 0,Y 445.952,Z 1255.989,A -85,B 0,C 180,E1 14832.107,E2 14832.107} C_VEL
LIN {X 0,Y 443.238,Z 1273.123,A -85,B 0,C 180,E1 14842.134,E2 14842.134} C_VEL
LIN {X 0,Y 443.38,Z 1276.979,A -85,B 0,C 180,E1 14850.98,E2 14850.98} C_VEL
LIN {X 0,Y 443.441,Z 1270.637,A -85,B 0,C 180,E1 14859.846,E2 14859.846} C_VEL
LIN {X 0,Y 446.356,Z 1252.12,A -85,B 0,C 180,E1 14869.346,E2 14869.346} C_VEL
LIN {X 0,Y 455.551,Z 1218.212,A -85,B 0,C 180,E1 14879.27,E2 14879.27} C_VEL
LIN {X 0,Y 471.286,Z 1170.41,A -85,B 0,C 180,E1 14888.146,E2 14888.146} C_VEL
LIN {X 0,Y 490.909,Z 1111.447,A -85,B 0,C 180,E1 14895.278,E2 14895.278} C_VEL
LIN {X 0,Y 510.402,Z 1044.891,A -85,B 0,C 180,E1 14900.448,E2 14900.448} C_VEL
LIN {X 0,Y 524.735,Z 976.696,A -85,B 0,C 180,E1 14903.877,E2 14903.877} C_VEL
